# B&R Automation Studio project OpcUaSample410_BrbLibUa103 (part 3)

#### BrbLib.typ - Exported data types
```iecst
(********************************************************************
 * COPYRIGHT -- Bernecker + Rainer
 ********************************************************************
 * Library: BrbLib
 * File: BrbLib.typ
 * Author: niedermeierr
 * Created: June 11, 2013
 ********************************************************************
 * Data types of library BrbLib
 ********************************************************************)
(*Error numbers*)

TYPE
	BrbError_ENUM :
		(
		eBRB_ERR_OK := 0,
		eBRB_ERR_NULL_POINTER := 50000,
		eBRB_ERR_INVALID_PARAMETER := 50001,
		eBRB_ERR_NOT_ENABLED := 50002,
		eBRB_ERR_OVERFLOW := 50003,
		eBRB_ERR_DIVISION_BY_0 := 50004,
		eBRB_ERR_STRING_TOO_SHORT := 50005,
		eBRB_ERR_STRING_TOO_LONG := 50006,
		eBRB_ERR_BUSY := 65535
		);
END_TYPE

(*StepHandling*)

TYPE
	BrbStepHandlingCurrent_TYP : 	STRUCT
		nStepNr : DINT; (*Aktuelle Schrittnummer*)
		sStepText : STRING[nBRB_STEP_TEXT_CHAR_MAX]; (*Aktueller Schritttext*)
		bTimeoutElapsed : BOOL; (*1=Timeout abgelaufen*)
		nTimeoutContinueStep : DINT; (*Schrittnummer nach Timeout*)
	END_STRUCT;
	BrbStepHandlingStep_TYP : 	STRUCT
		nStepNr : DINT; (*Schrittnummer*)
		sStepText : STRING[nBRB_STEP_TEXT_CHAR_MAX]; (*Schritttext*)
		nCycleCount : UDINT; (*Zyklen*)
	END_STRUCT;
	BrbStepHandlingLog_TYP : 	STRUCT
		bClear : BOOL; (*Kommando zum Löschen der Protokollierung*)
		bStop : BOOL; (*Kommando zum Stoppen der Protokollierung*)
		Steps : ARRAY[0..nBRB_STEPLOG_STEPS_MAX]OF BrbStepHandlingStep_TYP; (*Protokollierung*)
	END_STRUCT;
	BrbStepHandlingIntern_TYP : 	STRUCT
		nStepNrOld : DINT; (*Alte Schrittnummer*)
		nCycleCount : UDINT; (*Aktueller Zykluszähler*)
		bLogOnNextCycle : BOOL; (*Flag bei Schrittwechsel*)
		fbTimeout : TON; (*Timeout-Fub*)
	END_STRUCT;
	BrbStepHandling_TYP : 	STRUCT
		Current : BrbStepHandlingCurrent_TYP; (*Daten zum aktuellen Schritt*)
		Log : BrbStepHandlingLog_TYP; (*Protokollierung*)
		Intern : BrbStepHandlingIntern_TYP; (*Interne Daten*)
	END_STRUCT;
	BrbStopWatch_TYP : 	STRUCT
		tStartTime : TIME; (*Start-Zeitstempel*)
		tStopTime : TIME; (*End-Zeitstempel*)
		nTimeDiff : UDINT; (*Berechnete Differenz*)
		sTimeDiff : STRING[24]; (*Differenz als Text*)
	END_STRUCT;
END_TYPE

(*TaskCommunication*)

TYPE
	BrbCallerStates_ENUM :
		(
		eBRB_CALLER_STATE_NOT_READY := -1, (*-1=Nicht bereit*)
		eBRB_CALLER_STATE_OK := 0, (*0=Bereit*)
		eBRB_CALLER_STATE_BUSY := 1 (*1=Besetzt*)
		);
	BrbCaller_TYP : 	STRUCT
		nCallerId : DINT; (*Task-ID*)
		bLock : BOOL; (*Semaphor-Flag*)
	END_STRUCT;
END_TYPE

(*VarHandling*)

TYPE
	BrbLineBreak_ENUM :
		( (*Angabe des Zeilenumbruchs*)
		eBRB_LINE_BREAK_CRLF, (*0=CarriageReturn+LineFeed*)
		eBRB_LINE_BREAK_CR, (*1=CarriageReturn*)
		eBRB_LINE_BREAK_LF (*2=LineFeed*)
		);
	BrbPvInfo_TYP : 	STRUCT
		sName : STRING[nBRB_PVNAME_CHAR_MAX]; (*Variablen-Name*)
		nAdr : UDINT; (*Variablen-Adresse*)
		nDataType : UDINT; (*Variablen-Datentyp*)
		nLen : UDINT; (*Variablen-Größe*)
		nDimension : UINT; (*Max. Array-Index*)
		nItemIndex : UINT; (*Index des Array- oder Struktur-Items*)
	END_STRUCT;
END_TYPE

(*FileHandling*)

TYPE
	BrbUsbDeviceListEntry_TYP : 	STRUCT
		sInterfaceName : STRING[nBRB_DEVICE_NAME_CHAR_MAX]; (*Schnittstellen-Name*)
		sDeviceName : STRING[nBRB_DEVICE_NAME_CHAR_MAX]; (*Schnittstellen-Name*)
		nNode : UDINT; (*Interne Node-Nummer*)
		nHandle : UDINT; (*Internes Handle*)
	END_STRUCT;
	BrbDirInfoFilter_ENUM :
		(
		eBRB_DIR_INFO_ONLY_FILES, (*0=Nur Dateien*)
		eBRB_DIR_INFO_ONLY_DIRS, (*1=Nur Verzeichnisse*)
		eBRB_DIR_INFO_FILES_AND_DIRS (*2=Dateien und Verzeichnisse*)
		);
	BrbFileSorting_ENUM :
		(
		eBRB_FILE_SORTING_NONE, (*0=Keine Sortierung*)
		eBRB_FILE_SORTING_ALPH_UP, (*1=Sortierung nach aufsteigendem Alphabet*)
		eBRB_FILE_SORTING_ALPH_DOWN, (*2=Sortierung nach aufsteigendem Alphabet*)
		eBRB_FILE_SORTING_OLDEST, (*3=Sortierung nach ältesten Dateien*)
		eBRB_FILE_SORTING_YOUNGEST, (*4=Sortierung nach jüngsten Dateien*)
		eBRB_FILE_SORTING_BIGGEST, (*5=Sortierung nach größten Dateien*)
		eBRB_FILE_SORTING_SMALLEST, (*6=Sortierung nach kleinsten Dateien*)
		eBRB_FILE_SORTING_USER (*7=Sortierung mit benutzerdefinierter Vergleichsfunktion*)
		);
	BrbReadDirListEntry_TYP : 	STRUCT
		sName : STRING[nBRB_FILE_NAME_CHAR_MAX]; (*Verzeichnis- oder Datei-Name*)
		dtDate : DATE_AND_TIME; (*Zeitstempel*)
		nSize : UDINT; (*Größe (0=Verzeichnis)*)
	END_STRUCT;
END_TYPE

(*Logger*)

TYPE
	BrbLogHierarchListEntry_TYP : 	STRUCT
		nRecordId : ArEventLogRecordIDType;
		nOriginRecordId : ArEventLogRecordIDType;
		nEventId : DINT;
		nSeverity : USINT;
		sObjectId : STRING[36];
		sDecription : STRING[512];
	END_STRUCT;
	BrbLogHierarchListSevFilter_ENUM :
		(
		eBRB_LOG_SEVERITY_FILTER_ALL := 0, (*Keine Filterung*)
		eBRB_LOG_SEVERITY_FILTER_SUCCESS := 1, (*Nur Erfolgs-Einträge*)
		eBRB_LOG_SEVERITY_FILTER_INFO := 2, (*Nur Info-Einträge*)
		eBRB_LOG_SEVERITY_FILTER_WARNING := 4, (*Nur Warnungs-Einträge*)
		eBRB_LOG_SEVERITY_FILTER_ERROR := 8 (*Nur Fehler-Einträge*)
		);
END_TYPE

(*TimeAndDate*)

TYPE
	BrbWeekdays_ENUM :
		( (*Wochentage*)
		eBRB_WD_SUNDAY, (*0=Sonntag*)
		eBRB_WD_MONDAY, (*1=Montag*)
		eBRB_WD_TUESDAY, (*2=Dienstag*)
		eBRB_WD_WEDNESDAY, (*3=Mittwoch*)
		eBRB_WD_THURSDAY, (*4=Donnerstag*)
		eBRB_WD_FRIDAY, (*5=Freitag*)
		eBRB_WD_SATURDAY (*6=Samstag*)
		);
	BrbTimeAndDateCompare_ENUM :
		(
		eBRB_TAD_COMPARE_YOUNGER,
		eBRB_TAD_COMPARE_YOUNGEREQUAL,
		eBRB_TAD_COMPARE_EQUAL,
		eBRB_TAD_COMPARE_OLDEREQUAL,
		eBRB_TAD_COMPARE_OLDER
		);
	BrbTimerSwitchParTimePoint_TYP : 	STRUCT  (*Schaltpunkt*)
		bActive : BOOL; (*1=Zeitpunkt ist aktiv*)
		dtsTimePoint : DTStructure; (*Zeitpunkt*)
		eSwitchType : BrbTimerSwitchType_ENUM; (*Typ der Schaltung (Aus, An, Umschalten, Puls)*)
	END_STRUCT;
	BrbTimerSwitchPar_TYP : 	STRUCT  (*Parameter der Zeitschaltuhr*)
		eMode : BrbTimerSwitchMode_ENUM; (*Modus der Schaltung (Sekunde, Minute, Stunde...)*)
		TimePoint : ARRAY[0..nBRB_TIMERSWITCH_POINT_INDEX_MAX]OF BrbTimerSwitchParTimePoint_TYP; (*Liste der Schaltpunkte*)
	END_STRUCT;
	BrbTimerSwitchType_ENUM :
		( (*Typ der Schaltung*)
		eBRB_TIMERSWITCH_TYPE_OFF, (*0 = Aus*)
		eBRB_TIMERSWITCH_TYPE_ON, (*1 = An*)
		eBRB_TIMERSWITCH_TYPE_TOGGLE, (*2 = Umschalten*)
		eBRB_TIMERSWITCH_TYPE_IMPULSE (*3 = Puls*)
		);
	BrbTimerSwitchMode_ENUM :
		( (*Modus der Schaltung*)
		eBRB_TIMERSWITCH_MODE_MONTH, (*0=Monat*)
		eBRB_TIMERSWITCH_MODE_WEEK, (*1=Woche*)
		eBRB_TIMERSWITCH_MODE_DAY, (*2=Tag*)
		eBRB_TIMERSWITCH_MODE_HOUR, (*3=Stunde*)
		eBRB_TIMERSWITCH_MODE_MINUTE, (*4=Minute*)
		eBRB_TIMERSWITCH_MODE_SECOND (*5=Sekunde*)
		);
	BrbTimerSwitchWeekdays_ENUM :
		( (*Wochentage*)
		eBRB_TIMERSWITCH_WD_SUNDAY, (*0=Sonntag*)
		eBRB_TIMERSWITCH_WD_MONDAY, (*1=Montag*)
		eBRB_TIMERSWITCH_WD_TUESDAY, (*2=Dienstag*)
		eBRB_TIMERSWITCH_WD_WEDNESDAY, (*3=Mittwoch*)
		eBRB_TIMERSWITCH_WD_THURSDAY, (*4=Donnerstag*)
		eBRB_TIMERSWITCH_WD_FRIDAY, (*5=Freitag*)
		eBRB_TIMERSWITCH_WD_SATURDAY (*6=Samstag*)
		);
END_TYPE

(*BigDataTypes*)

TYPE
	BrbUint64_TYP : 	STRUCT
		nLow : UDINT; (*Niederwertige Bits*)
		nHigh : UDINT; (*Höherwertige Bits*)
	END_STRUCT;
	BrbInt64_TYP : 	STRUCT
		nLow : UDINT; (*Niederwertige Bits*)
		nHigh : UDINT; (*Höherwertige Bits*)
	END_STRUCT;
	BrbDt64Operator_ENUM :
		(
		eBRB_DT64_OPERATOR_ADD,
		eBRB_DT64_OPERATOR_SUBTRACT,
		eBRB_DT64_OPERATOR_MULTIPLY,
		eBRB_DT64_OPERATOR_DIVIDE
		);
END_TYPE

(*Memory*)

TYPE
	BrbMemListManagement_Typ : 	STRUCT
		pList : UDINT; (*Adresse des Array-Anfangs*)
		nEntryLength : UDINT; (*Größe eines Eintrags*)
		nIndexMax : UDINT; (*Maximaler Index des Arrays*)
		nEntryCount : UDINT; (*Momentane Anzahl der gültigen Eintrage*)
	END_STRUCT;
END_TYPE

(*Math*)

TYPE
	BrbRound_ENUM :
		(
		eBRB_ROUND_APPROP, (*Rundung gemäss letzter Stelle(n), Grenze bei 5*)
		eBRB_ROUND_UP, (*Aufrundung*)
		eBRB_ROUND_DOWN (*Abrundung*)
		);
END_TYPE

(*Random*)

TYPE
	BrbRandomString_ENUM :
		(
		eBRB_RANDOM_STRING_NUMBERS := 1, (*Zahler*)
		eBRB_RANDOM_STRING_UPPER_LETTERS := 2, (*Großbuchstaben*)
		eBRB_RANDOM_STRING_LOWER_LETTERS := 4, (*Kleinbuchstaben*)
		eBRB_RANDOM_STRING_SPACE := 8, (*Leerzeichen*)
		eBRB_RANDOM_STRING_PUNCTUATION := 16, (*Satzzeichen*)
		eBRB_RANDOM_STRING_SYMBOLS := 32, (*Symbole*)
		eBRB_RANDOM_STRING_CONTROLCHARS := 64 (*Steuerzeichen*)
		);
END_TYPE

(*IpAndSubnet*)

TYPE
	BrbIpAdrType_ENUM :
		( (*Ip-Adress-Typen*)
		eBRB_IP_ADR_TYPE_UNKNOWN, (*Unbekannte oder ungültige Adresse*)
		eBRB_IP_ADR_TYPE_NETWORK, (*Netzwerk-Adresse*)
		eBRB_IP_ADR_TYPE_HOST, (*Teilnehmer-Adresse*)
		eBRB_IP_ADR_TYPE_BROADCAST (*Broadcast-Adresse*)
		);
END_TYPE

(*Additional*)

TYPE
	BrbCompilerVersion_TYP : 	STRUCT
		bValid : BOOL; (*1=Version konnte ausgelesen werden*)
		nMajor : INT; (*Haupt-Versionsnummer*)
		nMinor : INT; (*Unter-Versionsnummer*)
		nPatch : INT; (*Patch-Versionsnummer*)
		nTotal : DINT; (*Komplette Versionnummer*)
		sText : STRING[10]; (*Versionsnummer als Text*)
	END_STRUCT;
END_TYPE
```

#### BrbLib.var - Exported constants
```iecst
(********************************************************************
 * COPYRIGHT -- Bernecker + Rainer
 ********************************************************************
 * Library: BrbLib
 * File: BrbLib.var
 * Author: niedermeierr
 * Created: June 11, 2013
 ********************************************************************
 * Constants of library BrbLib
 ********************************************************************)
(*General*)
VAR CONSTANT
	nBRB_USINT_MAX : USINT := 255; (*Maximal-Wert eines USINT*)
	nBRB_UINT_MAX : UINT := 65535; (*Maximal-Wert eines UINT*)
	nBRB_UDINT_MAX : UDINT := 4294967295; (*Maximal-Wert eines UDINT*)
	nBRB_SINT_MIN : SINT := -128; (*Minimal-Wert eines SINT*)
	nBRB_SINT_MAX : SINT := 127; (*Maximal-Wert eines SINT*)
	nBRB_INT_MIN : INT := -32768; (*Minimal-Wert eines INT*)
	nBRB_INT_MAX : INT := 32767; (*Maximal-Wert eines INT*)
	nBRB_DINT_MIN : DINT := -2147483648; (*Minimal-Wert eines DINT*)
	nBRB_DINT_MAX : DINT := 2147483647; (*Maximal-Wert eines DINT*)
	nBRB_BITS_PER_BYTE : USINT := 8; (*Anzahl Bits/Byte*)
	sBRB_STX : ARRAY[0..1] OF USINT := [2,0]; (*Start of Text*)
	sBRB_ETX : ARRAY[0..1] OF USINT := [3,0]; (*End of Text*)
	sBRB_TAB : ARRAY[0..1] OF USINT := [9,0]; (*Tabulator*)
	sBRB_LF : ARRAY[0..1] OF USINT := [10,0]; (*LineFeed = Vorschub*)
	sBRB_LFCR : ARRAY[0..2] OF USINT := [10,13,0]; (*LineFeed + CarriageReturn*)
	sBRB_CR : ARRAY[0..1] OF USINT := [13,0]; (*CarriageReturn = Wagenrücklauf*)
	sBRB_CRLF : ARRAY[0..2] OF USINT := [13,10,0]; (*CarriageReturn + LineFeed*)
	sBRB_QM : ARRAY[0..1] OF USINT := [34,0]; (*QuotationMark = Anführungszeichen*)
	sBRB_WC_TAB : ARRAY[0..1] OF UINT := [9,0]; (*Tabulator*)
	sBRB_WC_LF : ARRAY[0..1] OF UINT := [10,0]; (*LineFeed = Vorschub*)
	sBRB_WC_LFCR : ARRAY[0..2] OF UINT := [10,13,0]; (*LineFeed + CarriageReturn*)
	sBRB_WC_CR : ARRAY[0..1] OF UINT := [13,0]; (*CarriageReturn = Wagenrücklauf*)
	sBRB_WC_CRLF : ARRAY[0..2] OF UINT := [13,10,0]; (*CarriageReturn + LineFeed*)
	sBRB_WC_QM : ARRAY[0..1] OF UINT := [34,0]; (*QuotationMark = Anführungszeichen*)
	nBRB_URL_CHAR_MAX : UINT := 300; (*Zeichenanzahl einer URL*)
END_VAR
(*StepHandling*)
VAR CONSTANT
	nBRB_STEP_TEXT_CHAR_MAX : UINT := 50; (*Zeichenanzahl eines Schritt-Textes*)
	nBRB_STEPLOG_STEPS_MAX : UINT := 20; (*Max. Index der Protokollierung*)
END_VAR
(*VarHandling*)
VAR CONSTANT
	nBRB_FILE_LINES_CHAR_MAX : UINT := 50000; (*Zeichenanzahl einer Datei-Zeile*)
	nBRB_PVNAME_CHAR_MAX : UINT := 520; (*Zeichenanzahl eines Prozess-Variablen*)
END_VAR
(*FileHandling*)
VAR CONSTANT
	nBRB_DEVICE_NAME_CHAR_MAX : UDINT := 32; (*Zeichenanzahl eines Laufwerk-Namens*)
	nBRB_FILE_NAME_CHAR_MAX : UDINT := 259; (*Zeichenanzahl eines Datei-Namens*)
	nBRB_USB_DEVICE_LIST_INDEX_MAX : UINT := 5; (*Anzahl der Usb-Devices*)
	nBRB_FILTER_ALL_CHAR_MAX : UDINT := 200; (*Zeichenanzahl einer gesamten Filterangabe*)
	nBRB_FILTER_SINGLE_CHAR_MAX : UDINT := 20; (*Zeichenanzahl einer einzelnen Filterangabe*)
	nBRB_FILTER_SINGLE_INDEX_MAX : UDINT := 10; (*Max. Index der Filterrangaben*)
END_VAR
(*BigDataTypes*)
VAR CONSTANT
	nBRB_UINT64_CHAR_MAX : UINT := 21; (*Zeichenanzahl eines Uint64 (inkl. Null-Terminierung)*)
	nBRB_INT64_CHAR_MAX : UINT := 21; (*Zeichenanzahl eines Int64 (inkl. Null-Terminierung)*)
END_VAR
(*TimeAndDate*)
VAR CONSTANT
	nBRB_HOURS_PER_DAY : UDINT := 24; (*Stunden pro Tag*)
	nBRB_MINUTES_PER_HOUR : UDINT := 60; (*Minuten pro Stunde*)
	nBRB_SECONDS_PER_HOUR : UDINT := 3600; (*Sekunden pro Stunde*)
	nBRB_SECONDS_PER_DAY : UDINT := 86400; (*Sekunden pro Tag*)
	nBRB_SECONDS_PER_MINUTE : UDINT := 60; (*Sekunden pro Minute*)
	nBRB_MILLISECONDS_PER_SECOND : UDINT := 1000; (*Millisekunden pro Sekunde*)
	nBRB_MILLISECONDS_PER_MINUTE : UDINT := 60000; (*Millisekunden pro Minute*)
	nBRB_MILLISECONDS_PER_HOUR : UDINT := 3600000; (*Millisekunden pro Stunde*)
	nBRB_MILLISECONDS_PER_DAY : UDINT := 86400000; (*Millisekunden pro Tag*)
	nBRB_TIME_TEXT_CHAR_MAX : USINT := 24; (*Zeichenanzahl eines Zeitstempels*)
	nBRB_TIMERSWITCH_POINT_INDEX_MAX : UINT := 15; (*Maximaler Index der Zeitpunkt-Liste für die Zeitschaltuhr*)
END_VAR
(*Math*)
VAR CONSTANT
	rBRB_FACTOR_RAD_TO_DEG : REAL := 57.29578; (*Umrechnungsfaktor Bogenmass zu Grad*)
	rBRB_FACTOR_DEG_TO_RAD : REAL := 0.01745329; (*Umrechnungsfaktor Grad zu Bogenmass*)
	rBRB_DEGREE_0 : REAL := 0.0; (*0°*)
	rBRB_DEGREE_90 : REAL := 90.0; (*90°*)
	rBRB_DEGREE_180 : REAL := 180.0; (*180°*)
	rBRB_DEGREE_270 : REAL := 270.0; (*270°*)
	rBRB_DEGREE_360 : REAL := 360.0; (*360°*)
END_VAR
(*IpAndSubnet*)
VAR CONSTANT
	nBRB_IP_ADR_CHAR_MAX : UINT := 16; (*Anzahl der Zeichen einer IP-Adresse*)
END_VAR
```

#### AnsiCFunc.h
```c
/********************************************************************
 * COPYRIGHT -- Bernecker + Rainer
 ********************************************************************
 * Package: Global
 * File: AnsiCFunc.h
 * Author: niedermeierr
 * Created: April 22, 2008
 *******************************************************************/

#include <bur/plctypes.h>

/*
 * stdlib.h
 *
 * Definitions for common types, variables, and functions.
 */

// NOLINTBEGIN(bugprone-reserved-identifier, cert-dcl37-c, cppcoreguidelines-avoid-non-const-global-variables, clang-diagnostic-reserved-identifier)
#ifndef _STDLIB_H_
#define _STDLIB_H_

#include "_ansi.h"

#define __need_size_t
#define __need_wchar_t
#include <stddef.h>

#include <sys/reent.h>
#include <machine/stdlib.h>
#ifndef __STRICT_ANSI__
#include <alloca.h>
#endif

_BEGIN_STD_C

typedef struct
{
  int quot; /* quotient */
  int rem; /* remainder */
} div_t;

typedef struct
{
  long quot; /* quotient */
  long rem; /* remainder */
} ldiv_t;

#ifndef __STRICT_ANSI__
typedef struct
{
  long long int quot; /* quotient */
  long long int rem; /* remainder */
} lldiv_t;
#endif

#ifndef NULL
#define NULL 0
#endif

#define EXIT_FAILURE 1
#define EXIT_SUCCESS 0

#define RAND_MAX __RAND_MAX

extern __IMPORT int __mb_cur_max;

#define MB_CUR_MAX __mb_cur_max

_VOID	_EXFUN(abort,(_VOID) _ATTRIBUTE ((noreturn)));
int	_EXFUN(abs,(int));
int	_EXFUN(atexit,(_VOID (*__func)(_VOID)));
//double	_EXFUN(atof,(const char *__nptr));
#ifndef __STRICT_ANSI__
float	_EXFUN(atoff,(const char *__nptr));
#endif
//int	_EXFUN(atoi,(const char *__nptr));
int	_EXFUN(_atoi_r,(struct _reent *, const char *__nptr));
long	_EXFUN(atol,(const char *__nptr));
long	_EXFUN(_atol_r,(struct _reent *, const char *__nptr));
_PTR	_EXFUN(bsearch,(const _PTR __key,
		       const _PTR __base,
		       size_t __nmemb,
		       size_t __size,
		       int _EXPARM(_compar,(const _PTR, const _PTR))));
_PTR	_EXFUN(calloc,(size_t __nmemb, size_t __size));
div_t	_EXFUN(div,(int __numer, int __denom));
_VOID	_EXFUN(exit,(int __status) _ATTRIBUTE ((noreturn)));
_VOID	_EXFUN(free,(_PTR));
char *  _EXFUN(getenv,(const char *__string));
char *	_EXFUN(_getenv_r,(struct _reent *, const char *__string));
#ifdef __CYGWIN__
const char *_EXFUN(getprogname,(void));
#endif
char *	_EXFUN(_findenv,(_CONST char *, int *));
char *	_EXFUN(_findenv_r,(struct _reent *, _CONST char *, int *));
long	_EXFUN(labs,(long));
ldiv_t	_EXFUN(ldiv,(long __numer, long __denom));
_PTR	_EXFUN(malloc,(size_t __size));
int	_EXFUN(mblen,(const char *, size_t));
int	_EXFUN(_mblen_r,(struct _reent *, const char *, size_t, _mbstate_t *));
int	_EXFUN(mbtowc,(wchar_t *, const char *, size_t));
int	_EXFUN(_mbtowc_r,(struct _reent *, wchar_t *, const char *, size_t, _mbstate_t *));
int	_EXFUN(wctomb,(char *, wchar_t));
int	_EXFUN(_wctomb_r,(struct _reent *, char *, wchar_t, _mbstate_t *));
size_t	_EXFUN(mbstowcs,(wchar_t *, const char *, size_t));
size_t	_EXFUN(_mbstowcs_r,(struct _reent *, wchar_t *, const char *, size_t, _mbstate_t *));
size_t	_EXFUN(wcstombs,(char *, const wchar_t *, size_t));
size_t	_EXFUN(_wcstombs_r,(struct _reent *, char *, const wchar_t *, size_t, _mbstate_t *));
#ifndef __STRICT_ANSI__
#ifndef _REENT_ONLY
int     _EXFUN(mkstemp,(char *));
char *  _EXFUN(mktemp,(char *));
#endif
#endif
_VOID	_EXFUN(qsort,(_PTR __base, size_t __nmemb, size_t __size, int(*_compar)(const _PTR, const _PTR)));
int	_EXFUN(rand,(_VOID));
_PTR	_EXFUN(realloc,(_PTR __r, size_t __size));
#ifdef __CYGWIN__
void	_EXFUN(setprogname,(const char *));
#endif
_VOID	_EXFUN(srand,(unsigned __seed));
double	_EXFUN(strtod,(const char *__n, char **__end_PTR));
double	_EXFUN(_strtod_r,(struct _reent *,const char *__n, char **__end_PTR));
float	_EXFUN(strtof,(const char *__n, char **__end_PTR));
#ifndef __STRICT_ANSI__
/* the following strtodf interface is deprecated...use strtof instead */
# ifndef strtodf
#  define strtodf strtof
# endif
#endif
long	_EXFUN(strtol,(const char *__n, char **__end_PTR, int __base));
long	_EXFUN(_strtol_r,(struct _reent *,const char *__n, char **__end_PTR, int __base));
unsigned long _EXFUN(strtoul,(const char *__n, char **__end_PTR, int __base));
unsigned long _EXFUN(_strtoul_r,(struct _reent *,const char *__n, char **__end_PTR, int __base));

int	_EXFUN(system,(const char *__string));

#ifndef __STRICT_ANSI__
long    _EXFUN(a64l,(const char *__input));
char *  _EXFUN(l64a,(long __input));
char *  _EXFUN(_l64a_r,(struct _reent *,long __input));
int	_EXFUN(on_exit,(_VOID (*__func)(int, _PTR),_PTR __arg));
_VOID	_EXFUN(_Exit,(int __status) _ATTRIBUTE ((noreturn)));
int	_EXFUN(putenv,(const char *__string));
int	_EXFUN(_putenv_r,(struct _reent *, const char *__string));
int	_EXFUN(setenv,(const char *__string, const char *__value, int __overwrite));
int	_EXFUN(_setenv_r,(struct _reent *, const char *__string, const char *__value, int __overwrite));

char *	_EXFUN(gcvt,(double,int,char *));
char *	_EXFUN(gcvtf,(float,int,char *));
char *	_EXFUN(fcvt,(double,int,int *,int *));
char *	_EXFUN(fcvtf,(float,int,int *,int *));
char *	_EXFUN(ecvt,(double,int,int *,int *));
char *	_EXFUN(ecvtbuf,(double, int, int*, int*, char *));
char *	_EXFUN(fcvtbuf,(double, int, int*, int*, char *));
char *	_EXFUN(ecvtf,(float,int,int *,int *));
char *	_EXFUN(dtoa,(double, int, int, int *, int*, char**));
int	_EXFUN(rand_r,(unsigned *__seed));

double _EXFUN(drand48,(_VOID));
double _EXFUN(_drand48_r,(struct _reent *));
double _EXFUN(erand48,(unsigned short [3]));
double _EXFUN(_erand48_r,(struct _reent *, unsigned short [3]));
long   _EXFUN(jrand48,(unsigned short [3]));
long   _EXFUN(_jrand48_r,(struct _reent *, unsigned short [3]));
_VOID  _EXFUN(lcong48,(unsigned short [7]));
_VOID  _EXFUN(_lcong48_r,(struct _reent *, unsigned short [7]));
long   _EXFUN(lrand48,(_VOID));
long   _EXFUN(_lrand48_r,(struct _reent *));
long   _EXFUN(mrand48,(_VOID));
long   _EXFUN(_mrand48_r,(struct _reent *));
long   _EXFUN(nrand48,(unsigned short [3]));
long   _EXFUN(_nrand48_r,(struct _reent *, unsigned short [3]));
unsigned short *
       _EXFUN(seed48,(unsigned short [3]));
unsigned short *
       _EXFUN(_seed48_r,(struct _reent *, unsigned short [3]));
_VOID  _EXFUN(srand48,(long));
_VOID  _EXFUN(_srand48_r,(struct _reent *, long));
long long _EXFUN(atoll,(const char *__nptr));
long long _EXFUN(_atoll_r,(struct _reent *, const char *__nptr));
long long _EXFUN(llabs,(long long));
lldiv_t	_EXFUN(lldiv,(long long __numer, long long __denom));
long long _EXFUN(strtoll,(const char *__n, char **__end_PTR, int __base));
long long _EXFUN(_strtoll_r,(struct _reent *, const char *__n, char **__end_PTR, int __base));
unsigned long long _EXFUN(strtoull,(const char *__n, char **__end_PTR, int __base));
unsigned long long _EXFUN(_strtoull_r,(struct _reent *, const char *__n, char **__end_PTR, int __base));

#ifndef __CYGWIN__
_VOID	_EXFUN(cfree,(_PTR));
#else
char *	_EXFUN(realpath,(const char *, char *));
void	_EXFUN(unsetenv,(const char *__string));
void	_EXFUN(_unsetenv_r,(struct _reent *, const char *__string));
int	_EXFUN(random,(_VOID));
long	_EXFUN(srandom,(unsigned __seed));
char *  _EXFUN(ptsname, (int));
int     _EXFUN(grantpt, (int));
int     _EXFUN(unlockpt,(int));
#endif

#endif /* ! __STRICT_ANSI__ */

char *	_EXFUN(_dtoa_r,(struct _reent *, double, int, int, int *, int*, char**));
#ifndef __CYGWIN__
_PTR	_EXFUN(_malloc_r,(struct _reent *, size_t));
_PTR	_EXFUN(_calloc_r,(struct _reent *, size_t, size_t));
_VOID	_EXFUN(_free_r,(struct _reent *, _PTR));
_PTR	_EXFUN(_realloc_r,(struct _reent *, _PTR, size_t));
_VOID	_EXFUN(_mstats_r,(struct _reent *, char *));
#endif
int	_EXFUN(_system_r,(struct _reent *, const char *));

_VOID	_EXFUN(__eprintf,(const char *, const char *, unsigned int, const char *));

#ifdef __CYGWIN__
#undef _malloc_r
#define _malloc_r(r, s) malloc (s)
#undef _free_r
#define _free_r(r, p) free (p)
#undef _realloc_r
#define _realloc_r(r, p, s) realloc (p, s)
#undef _calloc_r
#define _calloc_r(r, s1, s2) calloc (s1, s2);
#undef _memalign_r
#define _memalign_r(r, s1, s2) memalign (s1, s2);
#undef _mallinfo_r
#define _mallinfo_r(r) mallinfo ()
#undef _malloc_stats_r
#define _malloc_stats_r(r) malloc_stats ()
#undef _mallopt_r
#define _mallopt_r(i1, i2) mallopt (i1, i2)
#undef _malloc_usable_size_r
#define _malloc_usable_size_r(r, p) malloc_usable_size (p)
#undef _valloc_r
#define _valloc_r(r, s) valloc (s)
#undef _pvalloc_r
#define _pvalloc_r(r, s) pvalloc (s)
#undef _malloc_trim_r
#define _malloc_trim_r(r, s) malloc_trim (s)
#undef _mstats_r
#define _mstats_r(r, p) mstats (p)
#endif

_END_STD_C

#endif /* _STDLIB_H_ */
// NOLINTEND(bugprone-reserved-identifier, cert-dcl37-c, cppcoreguidelines-avoid-non-const-global-variables, clang-diagnostic-reserved-identifier)
```

#### Package Logical/Libraries/BrbLib/StepHandling - Schrittketten-Behandlung

#### BrbStartStepTimeout.c
```c
/********************************************************************
 * COPYRIGHT -- Bernecker + Rainer
 ********************************************************************
 * Library: BrbLib
 * File: BrbStartStepTimeout.c
 * Author: niedermeierr
 * Created: June 11, 2013
 ********************************************************************
 * Implementation of library BrbLib
 ********************************************************************/

#include <bur/plctypes.h>
#ifdef __cplusplus
	extern "C"
	{
#endif

#include "BrbLib.h"

#ifdef __cplusplus
	};
#endif

 // NOLINTBEGIN(readability-*, bugprone-easily-swappable-parameters, clang-diagnostic-invalid-utf8, clang-diagnostic-invalid-source-encoding, clang-diagnostic-pointer-arith, clang-diagnostic-strict-prototypes, hicpp-uppercase-literal-suffix, cppcoreguidelines-*, performance-*)

/* Startet den Timeout-Zähler für eine Schrittkette */
unsigned short BrbStartStepTimeout(struct BrbStepHandling_TYP* pStepHandling, unsigned long nTimeout, signed long nContinueStep)
{
	// Prüfen, ob Timer schon abgelaufen ist
	if(pStepHandling->Intern.fbTimeout.Q == 0)
	{
		// Timer setzen und starten
		pStepHandling->Intern.fbTimeout.PT = (TIME)nTimeout;
		pStepHandling->Current.nTimeoutContinueStep = nContinueStep;
		pStepHandling->Intern.fbTimeout.IN = 1;
	}
	return 0;
}

// NOLINTEND(readability-*, bugprone-easily-swappable-parameters, clang-diagnostic-invalid-utf8, clang-diagnostic-invalid-source-encoding, clang-diagnostic-pointer-arith, clang-diagnostic-strict-prototypes, hicpp-uppercase-literal-suffix, cppcoreguidelines-*, performance-*)
```

#### BrbStartStopWatch.c
```c
/********************************************************************
 * COPYRIGHT -- Bernecker + Rainer
 ********************************************************************
 * Library: BrbLib
 * File: BrbStartStopWatch.c
 * Author: niedermeierr
 * Created: June 11, 2013
 ********************************************************************
 * Implementation of library BrbLib
 ********************************************************************/

#include <bur/plctypes.h>
#ifdef __cplusplus
	extern "C"
	{
#endif

#include "BrbLib.h"
#include <string.h>

#ifdef __cplusplus
	};
#endif

// NOLINTBEGIN(readability-*, bugprone-easily-swappable-parameters, clang-diagnostic-invalid-utf8, clang-diagnostic-invalid-source-encoding, clang-diagnostic-pointer-arith, clang-diagnostic-strict-prototypes, hicpp-uppercase-literal-suffix, cppcoreguidelines-*, performance-*)

/* Startet eine Stoppuhr */
plcbit BrbStartStopWatch(struct BrbStopWatch_TYP* pStopWatch)
{
	// Stoppuhr starten
	pStopWatch->tStartTime = clock_ms();
	pStopWatch->nTimeDiff = 0;
	memset(pStopWatch->sTimeDiff, 0, sizeof(pStopWatch->sTimeDiff));
	return 0;
}

// NOLINTEND(readability-*, bugprone-easily-swappable-parameters, clang-diagnostic-invalid-utf8, clang-diagnostic-invalid-source-encoding, clang-diagnostic-pointer-arith, clang-diagnostic-strict-prototypes, hicpp-uppercase-literal-suffix, cppcoreguidelines-*, performance-*)
```

#### BrbStepHandler.c
```c
/********************************************************************
 * COPYRIGHT -- Bernecker + Rainer
 ********************************************************************
 * Library: BrbLib
 * File: BrbStepHandler.c
 * Author: niedermeierr
 * Created: June 11, 2013
 ********************************************************************
 * Implementation of library BrbLib
 ********************************************************************/

#include <bur/plctypes.h>
#ifdef __cplusplus
	extern "C"
	{
#endif

#include "BrbLib.h"
#include <string.h>

#ifdef __cplusplus
	};
#endif

 // NOLINTBEGIN(readability-*, bugprone-easily-swappable-parameters, clang-diagnostic-invalid-utf8, clang-diagnostic-invalid-source-encoding, clang-diagnostic-pointer-arith, clang-diagnostic-strict-prototypes, hicpp-uppercase-literal-suffix, cppcoreguidelines-*, performance-*)

/* Behandelt Schrittketten (Protokollierung, Timeout usw.) */
signed long BrbStepHandler(struct BrbStepHandling_TYP* pStepHandling)
{
	// Muss der Schritt protokolliert werden?
	if(pStepHandling->Intern.bLogOnNextCycle == 1)
	{
		pStepHandling->Intern.bLogOnNextCycle = 0;
		// Ist Protokollierung gestoppt?
		if(pStepHandling->Log.bStop == 0)
		{
			// Zykluszähler merken
			pStepHandling->Log.Steps[0].nCycleCount = pStepHandling->Intern.nCycleCount;
			// Einträge um eins nach unten schieben
			memmove(&pStepHandling->Log.Steps[1], &pStepHandling->Log.Steps[0], sizeof(BrbStepHandlingStep_TYP)*(nBRB_STEPLOG_STEPS_MAX));
			// Aktuellen Eintrag reinkopieren
			pStepHandling->Log.Steps[0].nStepNr = pStepHandling->Intern.nStepNrOld;
			BrbStringCopy(pStepHandling->Log.Steps[0].sStepText, pStepHandling->Current.sStepText, sizeof(pStepHandling->Log.Steps[0].sStepText));
		}
		// Zykluszähler wieder auf 0 setzen
		pStepHandling->Intern.nCycleCount = 0;
	}
	// Hat sich der Schritt geändert?
	if(pStepHandling->Current.nStepNr != pStepHandling->Intern.nStepNrOld)
	{
		// Schritt beim nächsten Durchlauf protokollieren, weil dann erst der richtige Schritttext gesetzt ist
		pStepHandling->Intern.bLogOnNextCycle = 1;
	}
	// Zykluszähler erhöhen
	pStepHandling->Intern.nCycleCount++;
	// Aktuellen Schritt übernehmen
	pStepHandling->Intern.nStepNrOld = pStepHandling->Current.nStepNr;
	// Kommando zum Löschen der Protokollierung
	if(pStepHandling->Log.bClear == 1)
	{
		pStepHandling->Log.bClear = 0;
		// Den gesamten Aufzeichnungspuffer löschen
		memset(&pStepHandling->Log.Steps[0], 0, sizeof(pStepHandling->Log.Steps));
		pStepHandling->Intern.bLogOnNextCycle = 1;
	}
	// StepTimeout
	TON(&pStepHandling->Intern.fbTimeout);
	if(pStepHandling->Intern.fbTimeout.Q == 1)
	{
		// Timeout abgelaufen
		pStepHandling->Intern.fbTimeout.IN = 0;
		pStepHandling->Current.bTimeoutElapsed = 1;
	}
	return eBRB_ERR_OK;
}

 // NOLINTEND(readability-*, bugprone-easily-swappable-parameters, clang-diagnostic-invalid-utf8, clang-diagnostic-invalid-source-encoding, clang-diagnostic-pointer-arith, clang-diagnostic-strict-prototypes, hicpp-uppercase-literal-suffix, cppcoreguidelines-*, performance-*)
```

#### BrbStopStepTimeout.c
```c
/********************************************************************
 * COPYRIGHT -- Bernecker + Rainer
 ********************************************************************
 * Library: BrbLib
 * File: BrbStopStepTimeout.c
 * Author: niedermeierr
 * Created: June 11, 2013
 ********************************************************************
 * Implementation of library BrbLib
 ********************************************************************/

#include <bur/plctypes.h>
#ifdef __cplusplus
	extern "C"
	{
#endif

#include "BrbLib.h"

#ifdef __cplusplus
	};
#endif

// NOLINTBEGIN(readability-*, bugprone-easily-swappable-parameters, clang-diagnostic-invalid-utf8, clang-diagnostic-invalid-source-encoding, clang-diagnostic-pointer-arith, clang-diagnostic-strict-prototypes, hicpp-uppercase-literal-suffix, cppcoreguidelines-*, performance-*)

/* Stoppt den Timeout-Zähler für eine Schrittkette */
unsigned short BrbStopStepTimeout(struct BrbStepHandling_TYP* pStepHandling)
{
	// Timer stoppen
	pStepHandling->Intern.fbTimeout.IN = 0;
	return 0;
}

// NOLINTEND(readability-*, bugprone-easily-swappable-parameters, clang-diagnostic-invalid-utf8, clang-diagnostic-invalid-source-encoding, clang-diagnostic-pointer-arith, clang-diagnostic-strict-prototypes, hicpp-uppercase-literal-suffix, cppcoreguidelines-*, performance-*)
```

#### BrbStopStopWatch.c
```c
/********************************************************************
 * COPYRIGHT -- Bernecker + Rainer
 ********************************************************************
 * Library: BrbLib
 * File: BrbStopStopWatch.c
 * Author: niedermeierr
 * Created: June 11, 2013
 ********************************************************************
 * Implementation of library BrbLib
 ********************************************************************/

#include <bur/plctypes.h>
#ifdef __cplusplus
	extern "C"
	{
#endif

#include "BrbLib.h"
#include <string.h>

#ifdef __cplusplus
	};
#endif

// NOLINTBEGIN(readability-*, bugprone-easily-swappable-parameters, clang-diagnostic-invalid-utf8, clang-diagnostic-invalid-source-encoding, clang-diagnostic-pointer-arith, clang-diagnostic-strict-prototypes, hicpp-uppercase-literal-suffix, cppcoreguidelines-*, performance-*)

/* Stoppt eine Stoppuhr */
unsigned long BrbStopStopWatch(struct BrbStopWatch_TYP* pStopWatch)
{
	// Stoppuhr stoppen
	pStopWatch->tStopTime = clock_ms();
	pStopWatch->nTimeDiff = DiffT(pStopWatch->tStopTime, pStopWatch->tStartTime);
	memset(pStopWatch->sTimeDiff, 0, sizeof(pStopWatch->sTimeDiff));
	TIMEStructure TimeDiff;
	TIME_TO_TIMEStructure((TIME)pStopWatch->nTimeDiff, (UDINT)&TimeDiff);
	STRING sItoA[20];
	memset(sItoA, 0, sizeof(sItoA));
	if(TimeDiff.day < 10)
	{
		BrbStringCat((STRING*)pStopWatch->sTimeDiff, "0", sizeof(pStopWatch->sTimeDiff));
	}
	brsitoa((DINT)TimeDiff.day, (UDINT)&sItoA);
	BrbStringCat((STRING*)pStopWatch->sTimeDiff, sItoA, sizeof(pStopWatch->sTimeDiff));
	BrbStringCat((STRING*)pStopWatch->sTimeDiff, "d_", sizeof(pStopWatch->sTimeDiff));
	if(TimeDiff.hour < 10)
	{
		BrbStringCat((STRING*)pStopWatch->sTimeDiff, "0", sizeof(pStopWatch->sTimeDiff));
	}
	brsitoa((DINT)TimeDiff.hour, (UDINT)&sItoA);
	BrbStringCat((STRING*)pStopWatch->sTimeDiff, sItoA, sizeof(pStopWatch->sTimeDiff));
	BrbStringCat((STRING*)pStopWatch->sTimeDiff, "h_", sizeof(pStopWatch->sTimeDiff));
	if(TimeDiff.minute < 10)
	{
		BrbStringCat((STRING*)pStopWatch->sTimeDiff, "0", sizeof(pStopWatch->sTimeDiff));
	}
	brsitoa((DINT)TimeDiff.minute, (UDINT)&sItoA);
	BrbStringCat((STRING*)pStopWatch->sTimeDiff, sItoA, sizeof(pStopWatch->sTimeDiff));
	BrbStringCat((STRING*)pStopWatch->sTimeDiff, "m_", sizeof(pStopWatch->sTimeDiff));
	if(TimeDiff.second < 10)
	{
		BrbStringCat((STRING*)pStopWatch->sTimeDiff, "0", sizeof(pStopWatch->sTimeDiff));
	}
	brsitoa((DINT)TimeDiff.second, (UDINT)&sItoA);
	BrbStringCat((STRING*)pStopWatch->sTimeDiff, sItoA, sizeof(pStopWatch->sTimeDiff));
	BrbStringCat((STRING*)pStopWatch->sTimeDiff, "s_", sizeof(pStopWatch->sTimeDiff));
	if(TimeDiff.millisec < 10)
	{
		BrbStringCat((STRING*)pStopWatch->sTimeDiff, "00", sizeof(pStopWatch->sTimeDiff));
	}
	else if(TimeDiff.millisec < 100)
	{
		BrbStringCat((STRING*)pStopWatch->sTimeDiff, "0", sizeof(pStopWatch->sTimeDiff));
	}
	brsitoa((DINT)TimeDiff.millisec, (UDINT)&sItoA);
	BrbStringCat((STRING*)pStopWatch->sTimeDiff, sItoA, sizeof(pStopWatch->sTimeDiff));
	BrbStringCat((STRING*)pStopWatch->sTimeDiff, "ms", sizeof(pStopWatch->sTimeDiff));
	return pStopWatch->nTimeDiff;
}

// NOLINTEND(readability-*, bugprone-easily-swappable-parameters, clang-diagnostic-invalid-utf8, clang-diagnostic-invalid-source-encoding, clang-diagnostic-pointer-arith, clang-diagnostic-strict-prototypes, hicpp-uppercase-literal-suffix, cppcoreguidelines-*, performance-*)
```

#### Package Logical/Libraries/BrbLib/TaskCommunication - Task-Kommunikation

#### BrbClearCallerBox.c
```c
/********************************************************************
 * COPYRIGHT -- Bernecker + Rainer
 ********************************************************************
 * Library: BrbLib
 * File: BrbClearCallerBox.c
 * Author: niedermeierr
 * Created: June 11, 2013
 ********************************************************************
 * Implementation of library BrbLib
 ********************************************************************/

#include <bur/plctypes.h>
#ifdef __cplusplus
	extern "C"
	{
#endif

#include "BrbLib.h"
#include <string.h>

#ifdef __cplusplus
	};
#endif

// NOLINTBEGIN(readability-*, bugprone-easily-swappable-parameters, clang-diagnostic-invalid-utf8, clang-diagnostic-invalid-source-encoding, clang-diagnostic-pointer-arith, clang-diagnostic-strict-prototypes, hicpp-uppercase-literal-suffix, cppcoreguidelines-*, performance-*)

/* Setzt eine CallerBox komplett auf 0 */
unsigned short BrbClearCallerBox(unsigned long pCallerBox, unsigned long nSize)
{
	memset((USINT*)pCallerBox, 0, nSize);
	return eBRB_ERR_OK;
}

// NOLINTEND(readability-*, bugprone-easily-swappable-parameters, clang-diagnostic-invalid-utf8, clang-diagnostic-invalid-source-encoding, clang-diagnostic-pointer-arith, clang-diagnostic-strict-prototypes, hicpp-uppercase-literal-suffix, cppcoreguidelines-*, performance-*)
```

#### BrbClearDirectBox.c
```c
/********************************************************************
 * COPYRIGHT -- Bernecker + Rainer
 ********************************************************************
 * Library: BrbLib
 * File: BrbClearDirectBox.c
 * Author: niedermeierr
 * Created: June 11, 2013
 ********************************************************************
 * Implementation of library BrbLib
 ********************************************************************/

#include <bur/plctypes.h>
#ifdef __cplusplus
	extern "C"
	{
#endif

#include "BrbLib.h"
#include <string.h>

#ifdef __cplusplus
	};
#endif

// NOLINTBEGIN(readability-*, bugprone-easily-swappable-parameters, clang-diagnostic-invalid-utf8, clang-diagnostic-invalid-source-encoding, clang-diagnostic-pointer-arith, clang-diagnostic-strict-prototypes, hicpp-uppercase-literal-suffix, cppcoreguidelines-*, performance-*)

/* Setzt eine DirectBox komplett auf 0 */
unsigned short BrbClearDirectBox(unsigned long pDirectBox, unsigned long nSize)
{
	memset((USINT*)pDirectBox, 0, nSize);
	return eBRB_ERR_OK;
}

// NOLINTEND(readability-*, bugprone-easily-swappable-parameters, clang-diagnostic-invalid-utf8, clang-diagnostic-invalid-source-encoding, clang-diagnostic-pointer-arith, clang-diagnostic-strict-prototypes, hicpp-uppercase-literal-suffix, cppcoreguidelines-*, performance-*)
```

#### BrbSetCaller.c
```c
/********************************************************************
 * COPYRIGHT -- Bernecker + Rainer
 ********************************************************************
 * Library: BrbLib
 * File: BrbSetCaller.c
 * Author: niedermeierr
 * Created: June 11, 2013
 ********************************************************************
 * Implementation of library BrbLib
 ********************************************************************/

#include <bur/plctypes.h>
#ifdef __cplusplus
	extern "C"
	{
#endif

#include "BrbLib.h"

#ifdef __cplusplus
	};
#endif

// NOLINTBEGIN(readability-*, bugprone-easily-swappable-parameters, clang-diagnostic-invalid-utf8, clang-diagnostic-invalid-source-encoding, clang-diagnostic-pointer-arith, clang-diagnostic-strict-prototypes, hicpp-uppercase-literal-suffix, cppcoreguidelines-*, performance-*)

/* Versucht, die Reservierung für ein Task-Kommando zu erhalten */
BrbCallerStates_ENUM BrbSetCaller(struct BrbCaller_TYP* pCaller, signed long nCallerId)
{
	// Prüfung der Parameter
	if(pCaller == 0)
	{
		return eBRB_CALLER_STATE_NOT_READY;
	}
	// Prüfen, ob die CallerId gesetzt werden kann
	if((pCaller->nCallerId == 0) && (pCaller->bLock == 0))
	{
		// CallerId setzen
		pCaller->nCallerId = nCallerId;
		// Prüfen, ob der Aufruf von einer schnelleren Taskklasse unterbrochen wurde
		if((pCaller->nCallerId == nCallerId) && (pCaller->bLock == 0))
		{
			// CallerId konnte gesetzt werden
			pCaller->bLock = 1;
			return eBRB_CALLER_STATE_OK;
		}
		else
		{
			// Das Setzen wurde von einer schnelleren Taskklasse unterbrochen
			return eBRB_CALLER_STATE_BUSY;
		}
	}
	else if(pCaller->nCallerId == -1)
	{
		// Der Task ist noch nicht bereit
		return eBRB_CALLER_STATE_NOT_READY;
	}
	else
	{
		// Der Task ist schon reserviert
		return eBRB_CALLER_STATE_BUSY;
	}
}

// NOLINTEND(readability-*, bugprone-easily-swappable-parameters, clang-diagnostic-invalid-utf8, clang-diagnostic-invalid-source-encoding, clang-diagnostic-pointer-arith, clang-diagnostic-strict-prototypes, hicpp-uppercase-literal-suffix, cppcoreguidelines-*, performance-*)
```

#### Package Logical/Libraries/BrbLib/VarHandling - Variablen-Funktionen

#### BrbLoadVarAscii.c
```c
/********************************************************************
 * COPYRIGHT -- Bernecker + Rainer
 ********************************************************************
 * Library: BrbLib
 * File: BrbLoadVarAscii.c
 * Author: niedermeierr
 * Created: June 11, 2013
 ********************************************************************
 * Implementation of library BrbLib
 ********************************************************************/

#include <bur/plctypes.h>
#ifdef __cplusplus
	extern "C"
	{
#endif

#include "BrbLib.h"
#include <string.h>

#ifdef __cplusplus
	};
#endif

// NOLINTBEGIN(readability-*, bugprone-easily-swappable-parameters, clang-diagnostic-invalid-utf8, clang-diagnostic-invalid-source-encoding, clang-diagnostic-pointer-arith, clang-diagnostic-strict-prototypes, hicpp-uppercase-literal-suffix, cppcoreguidelines-*, performance-*)

// Eigene Enums und Typen
enum Steps_ENUM
{
	eSTEP_INIT,
	eSTEP_GET_DATAOBJ_INFO,
	eSTEP_DELETE_DATAOBJ_START,
	eSTEP_OPEN_FILE,
	eSTEP_CREATE_DATAOBJ,
	eSTEP_READ_FILE,
	eSTEP_CLOSE_FILE,
	eSTEP_READ_LINES,
	eSTEP_DELETE_DATAOBJ_END,
};

enum Datatypes_ENUM
{
	eDATATYPE_STRUCT,
	eDATATYPE_BOOL,
	eDATATYPE_SINT,
	eDATATYPE_INT,
	eDATATYPE_DINT,
	eDATATYPE_USINT,
	eDATATYPE_UINT,
	eDATATYPE_UDINT,
	eDATATYPE_REAL,
	eDATATYPE_STRING,
	eDATATYPE_DATE_AND_TIME = 11,
	eDATATYPE_TIME,
	eDATATYPE_STRUCT_ARRAY = 15
};

// Prototypen
STRING* SetToNextLine(STRING* pText, STRING* pTextEnd, STRING* pLineBreak);
STRING* ReadPvName(STRING* pText, STRING* pPvName, STRING* pTextEnd);
STRING* ReadPvValue(STRING* pText, STRING* pPvValue, STRING* pTextEnd);
void SetValue(BrbPvInfo_TYP* pPvInfo, STRING* pValue);

/* Lädt eine Ascii-Datei mit Variablen-Werten */
void BrbLoadVarAscii(struct BrbLoadVarAscii* inst) // NOLINT(readability-function-cognitive-complexity)
{
	// Prüfung der Parameter
	if(inst->pDevice == 0)
	{
		inst->nStatus = eBRB_ERR_NULL_POINTER;
		return;
	}
	if(inst->pFile == 0)
	{
		inst->nStatus = eBRB_ERR_NULL_POINTER;
		return;
	}

	switch(inst->eStep)
	{
		case eSTEP_INIT:
			// Fub initialisieren
			inst->nStatus = eBRB_ERR_BUSY;
			inst->nStatusIntern = 0;
			memset(&inst->fbDatObjInfo, 0, sizeof(inst->fbDatObjInfo));
			memset(&inst->fbDatObjDelete, 0, sizeof(inst->fbDatObjDelete));
			memset(&inst->fbFileOpen, 0, sizeof(inst->fbFileOpen));
			memset(&inst->fbDatObjCreate, 0, sizeof(inst->fbDatObjCreate));
			switch(inst->eLineBeak) // NOLINT(clang-diagnostic-switch-enum)
			{
				case eBRB_LINE_BREAK_CR:
					strcpy(inst->sLineBreak, "\r");
					break;
				case eBRB_LINE_BREAK_LF:
					strcpy(inst->sLineBreak, "\n");
					break;
				default:
					strcpy(inst->sLineBreak, "\r\n");
					break;
			}
			if(inst->nLinesToReadAtOneStep == 0)
			{
				// Wenn keine Anzahl angegeben ist, einen Defaultwert verwenden
				inst->nLinesToReadAtOneStep = 10;
			}
			inst->pTextStart = 0;
			inst->pTextEnd = 0;
			inst->pText = 0;
			inst->nLineCountRead = 0;
			memset(&inst->fbFileRead, 0, sizeof(inst->fbFileRead));
			memset(&inst->fbFileClose, 0, sizeof(inst->fbFileClose));
			inst->eStep = eSTEP_GET_DATAOBJ_INFO;
			break;

		case eSTEP_GET_DATAOBJ_INFO:
			// Prüfen, ob noch ein altes Datenobjekt vorhanden ist
			inst->nStatus = eBRB_ERR_BUSY;
			inst->fbDatObjInfo.enable = 1;
			inst->fbDatObjInfo.pName = (UDINT)&"LdPv123";
			DatObjInfo(&inst->fbDatObjInfo);
			if(inst->fbDatObjInfo.status == 0)
			{
				// Vorhanden -> löschen
				inst->eStep = eSTEP_DELETE_DATAOBJ_START;
			}
			else if(inst->fbDatObjInfo.status != eBRB_ERR_BUSY)
			{
				// Nicht vorhanden -> Datei öffnen
				inst->eStep = eSTEP_OPEN_FILE;
			}
			break;

		case eSTEP_DELETE_DATAOBJ_START:
			// Evtl. noch vorhandenes Datenobjekt löschen
			inst->nStatus = eBRB_ERR_BUSY;
			inst->fbDatObjDelete.enable = 1;
			inst->fbDatObjDelete.ident = inst->fbDatObjCreate.ident;
			DatObjDelete(&inst->fbDatObjDelete);
			if(inst->fbDatObjDelete.status == 0)
			{
				inst->eStep = eSTEP_OPEN_FILE;
			}
			else if(inst->fbDatObjDelete.status != eBRB_ERR_BUSY)
			{
				inst->nStatus = inst->fbFileOpen.status;
				inst->eStep = eSTEP_INIT;
			}
			break;

		case eSTEP_OPEN_FILE:
			// Datei öffnen
			inst->nStatus = eBRB_ERR_BUSY;
			inst->fbFileOpen.enable = 1;
			inst->fbFileOpen.pDevice = (UDINT)inst->pDevice;
			inst->fbFileOpen.pFile = (UDINT)inst->pFile;
			FileOpen(&inst->fbFileOpen);
			if(inst->fbFileOpen.status == 0)
			{
				inst->eStep = eSTEP_CREATE_DATAOBJ;
			}
			else if(inst->fbFileOpen.status != eBRB_ERR_BUSY)
			{
				inst->nStatus = inst->fbFileOpen.status;
				inst->eStep = eSTEP_INIT;
			}
			break;

		case eSTEP_CREATE_DATAOBJ:
			// Datenobjekt mit der Größe der Datei erzeugen
			inst->nStatus = eBRB_ERR_BUSY;
			inst->fbDatObjCreate.enable = 1;
			inst->fbDatObjCreate.grp = 0;
			inst->fbDatObjCreate.pName = (UDINT)&"LdPv123";
			inst->fbDatObjCreate.len = inst->fbFileOpen.filelen;
			inst->fbDatObjCreate.MemType = doTEMP;
			inst->fbDatObjCreate.Option = doNO_CS;
			inst->fbDatObjCreate.pCpyData = 0;
			DatObjCreate(&inst->fbDatObjCreate);
			if(inst->fbDatObjCreate.status == 0)
			{
				inst->pTextStart = (STRING*)inst->fbDatObjCreate.pDatObjMem;
				inst->pTextEnd = inst->pTextStart + inst->fbDatObjCreate.len;
				inst->pText = inst->pTextStart;
				inst->eStep = eSTEP_READ_FILE;
			}
			else if(inst->fbDatObjCreate.status != eBRB_ERR_BUSY)
			{
				// Fehler merken
				inst->nStatusIntern = inst->fbDatObjCreate.status;
				// Datei muß auf jeden Fall geschlossen werden
				inst->eStep = eSTEP_CLOSE_FILE;
			}
			break;

		case eSTEP_READ_FILE:
			// Datei in das Datenobjekt einlesen
			inst->nStatus = eBRB_ERR_BUSY;
			inst->fbFileRead.enable = 1;
			inst->fbFileRead.ident = inst->fbFileOpen.ident;
			inst->fbFileRead.offset = 0;
			inst->fbFileRead.pDest = inst->fbDatObjCreate.pDatObjMem;
			inst->fbFileRead.len = inst->fbFileOpen.filelen;
			FileRead(&inst->fbFileRead);
			if(inst->fbFileRead.status == 0)
			{
				inst->eStep = eSTEP_CLOSE_FILE;
			}
			else if(inst->fbFileRead.status != eBRB_ERR_BUSY)
			{
				// Fehler merken
				inst->nStatusIntern = inst->fbFileRead.status;
				// Datei muß auf jeden Fall geschlossen werden
				inst->eStep = eSTEP_CLOSE_FILE;
			}
			break;

		case eSTEP_CLOSE_FILE:
			// Datei schliessen
			inst->nStatus = eBRB_ERR_BUSY;
			inst->fbFileClose.enable = 1;
			inst->fbFileClose.ident = inst->fbFileOpen.ident;
			FileClose(&inst->fbFileClose);
			if(inst->fbFileClose.status == 0)
			{
				// Prüfen, ob vorher schon ein Fehler aufgetreten ist
				if(inst->nStatusIntern > 0)
				{
					// Datenobjekt muß auf jeden Fall gelöscht werden
					inst->eStep = eSTEP_DELETE_DATAOBJ_END;
				}
				else
				{
					inst->eStep = eSTEP_READ_LINES;
				}
			}
			else if(inst->fbFileClose.status != eBRB_ERR_BUSY)
			{
				// Prüfen, ob vorher schon ein Fehler aufgetreten ist
				if(inst->nStatusIntern > 0)
				{
					// Datenobjekt muß auf jeden Fall gelöscht werden
					inst->eStep = eSTEP_DELETE_DATAOBJ_END;
				}
				else
				{
					// Fehler merken
					inst->nStatusIntern = inst->fbFileClose.status;
					// Datenobjekt muß auf jeden Fall gelöscht werden
					inst->eStep = eSTEP_DELETE_DATAOBJ_END;
				}
			}
			break;

		case eSTEP_READ_LINES:
			inst->nStatus = eBRB_ERR_BUSY;
			inst->nLineCountRead = 0;
			do
			{
				if(BrbStringStartsWith(inst->pText, "//"))
				{
					// Kommentare werden überlesen
				}
				else
				{
					// Variable lesen
					BrbPvInfo_TYP PvInfo;
					memset(&PvInfo, 0, sizeof(PvInfo));
					STRING sPvValue[nBRB_PVNAME_CHAR_MAX];
					memset(&sPvValue, 0, sizeof(sPvValue));
					// Namen lesen
					inst->pText = ReadPvName(inst->pText, PvInfo.sName, inst->pTextEnd);
					if(inst->pText != 0)
					{
						// Wert lesen
						inst->pText = ReadPvValue(inst->pText, sPvValue, inst->pTextEnd);
						if(inst->pText != 0)
						{
							SetValue(&PvInfo, sPvValue);
						}
					}
				}
				// Auf den Anfang der nächsten Zeile springen
				inst->pText = SetToNextLine(inst->pText, inst->pTextEnd, (STRING*)&inst->sLineBreak);
				inst->nLineCountRead += 1;
				if((inst->pText >= inst->pTextEnd) || (inst->pText == 0))
				{
					// Ende der Datei erreicht -> Schleife verlassen
					inst->nLineCountRead = inst->nLinesToReadAtOneStep + 1;
					inst->eStep = eSTEP_DELETE_DATAOBJ_END;
					break;
				}
			}
			while(inst->nLineCountRead <= inst->nLinesToReadAtOneStep);
			break;

		case eSTEP_DELETE_DATAOBJ_END:
			// Datenobjekt löschen
			inst->nStatus = eBRB_ERR_BUSY;
			inst->fbDatObjDelete.enable = 1;
			inst->fbDatObjDelete.ident = inst->fbDatObjCreate.ident;
			DatObjDelete(&inst->fbDatObjDelete);
			if(inst->fbDatObjDelete.status != eBRB_ERR_BUSY)
			{
				if(inst->nStatusIntern > 0)
				{
					inst->nStatus = inst->nStatusIntern;
				}
				else
				{
					inst->nStatus = 0;
				}
				inst->eStep = eSTEP_INIT;
			}
			break;

	}
}

// Gibt die Adresse nach dem nächsten Zeilenumbruch zurück.
// 0, wenn es nicht gefunden wird.
STRING* SetToNextLine(STRING* pText, STRING* pTextEnd, STRING* pLineBreak)
{
	STRING* pResult = 0;
	if(pText != 0)
	{
		// Nach Zeilenumbruch suchen
		pResult = BrbStringGetAdrOf(pText, pLineBreak, (UDINT)(pTextEnd - pText));
		if(pResult >= pText)
		{
			// Gefunden -> CrLf überspringen
			pResult += 2;
		}
	}
	return pResult;
}

// Liest den Text bis zum nächsten = und gibt die Adresse danach zurück.
// 0, wenn es nicht gefunden wird.
STRING* ReadPvName(STRING* pText, STRING* pPvName, STRING* pTextEnd)
{
	STRING* pResult = 0;
	// Nach = suchen
	pResult = BrbStringGetAdrOf(pText, "=", (UDINT)(pTextEnd - pText));
	if(pResult >= pText)
	{
		// Gefunden -> Überspringen
		memcpy(pPvName, pText, (UDINT)(pResult - pText));
		pResult += 1;
	}
	return pResult;
}

// Liest den Text bis zum nächsten CrLf und gibt die Adresse zurück.
// 0, wenn es nicht gefunden wird.
STRING* ReadPvValue(STRING* pText, STRING* pPvValue, STRING* pTextEnd)
{
	STRING* pResult = 0;
	// Nach CrLf suchen
	pResult = BrbStringGetAdrOf(pText, "\r\n", (UDINT)(pTextEnd - pText));
	if(pResult >= pText)
	{

		// Gefunden -> Länge des Werts prüfen
		UDINT nLenValue = (UDINT)(pResult - pText);
		if(nLenValue >= nBRB_PVNAME_CHAR_MAX)
		{
			// Länge begrenzen
			nLenValue = nBRB_PVNAME_CHAR_MAX - 1;
		}
		// Wert kopieren
		memcpy(pPvValue, pText, nLenValue);
		// CrLf nicht überspringen (wird zum Erkennen der nächsten Zeile gebraucht)
	}
	return pResult;
}

// Setzt den Wert einer Pv als String.
void SetValue(BrbPvInfo_TYP* pPvInfo, STRING* pValue)
{
	UINT	nFuncStatus = 0;
	UDINT nLen = 0;
	STRING sItoA[20];
	memset(sItoA, 0, sizeof(sItoA));
	// Adresse der Variablen holen
	nFuncStatus = PV_xgetadr(pPvInfo->sName, &pPvInfo->nAdr, &nLen);
	if(nFuncStatus == 0)
	{
		// Datentyp der Variable holen
		nFuncStatus = PV_ninfo(pPvInfo->sName, &pPvInfo->nDataType, &pPvInfo->nLen, &pPvInfo->nDimension);
		if(nFuncStatus == 0)
		{
			// Wert in Datentyp wandeln und an der Adresse setzen
			switch(pPvInfo->nDataType)
			{
				case eDATATYPE_BOOL:
					{
						DINT nValue = brsatoi((UDINT)pValue);
						*(BOOL*)pPvInfo->nAdr = (BOOL)nValue;
					}
					break;

				case eDATATYPE_SINT:
					{
						DINT nValue = brsatoi((UDINT)pValue);
						*(SINT*)pPvInfo->nAdr = (SINT)nValue;
					}
					break;

				case eDATATYPE_INT:
					{
						DINT nValue = brsatoi((UDINT)pValue);
						*(INT*)pPvInfo->nAdr = (INT)nValue;
					}
					break;

				case eDATATYPE_DINT:
					{
						DINT nValue = brsatoi((UDINT)pValue);
						*(DINT*)pPvInfo->nAdr = (DINT)nValue;
					}
					break;

				case eDATATYPE_USINT:
					{
						DINT nValue = brsatoi((UDINT)pValue);
						*(USINT*)pPvInfo->nAdr = (USINT)nValue;
					}
					break;

				case eDATATYPE_UINT:
					{
						DINT nValue = brsatoi((UDINT)pValue);
						*(UINT*)pPvInfo->nAdr = (UINT)nValue;
					}
					break;

				case eDATATYPE_UDINT:
					{
						UDINT nValue = BrbAsciiToUdint(pValue);
						*(UDINT*)pPvInfo->nAdr = (UDINT)nValue;
					}
					break;

				case eDATATYPE_REAL:
					{
						REAL rValue = brsatof((UDINT)pValue);
						*(REAL*)pPvInfo->nAdr = (REAL)rValue;
					}
					break;

				case eDATATYPE_STRING:
					{
						strcpy((STRING*)pPvInfo->nAdr, pValue); // NOLINT(clang-analyzer-security.insecureAPI.strcpy)
					}
					break;

				case eDATATYPE_DATE_AND_TIME:
					{
						UDINT nValue = BrbAsciiToUdint(pValue);
						*(UDINT*)pPvInfo->nAdr = (UDINT)nValue;
					}
					break;

				case eDATATYPE_TIME:
					{
						DINT nValue = brsatoi((UDINT)pValue);
						*(DINT*)pPvInfo->nAdr = (DINT)nValue;
					}
					break;

			}
		}
	}
}

// NOLINTEND(readability-*, bugprone-easily-swappable-parameters, clang-diagnostic-invalid-utf8, clang-diagnostic-invalid-source-encoding, clang-diagnostic-pointer-arith, clang-diagnostic-strict-prototypes, hicpp-uppercase-literal-suffix, cppcoreguidelines-*, performance-*)
```

#### BrbLoadVarBin.c
```c
/********************************************************************
 * COPYRIGHT -- Bernecker + Rainer
 ********************************************************************
 * Library: BrbLib
 * File: BrbLoadVarBin.c
 * Author: niedermeierr
 * Created: June 11, 2013
 ********************************************************************
 * Implementation of library BrbLib
 ********************************************************************/

#include <bur/plctypes.h>
#ifdef __cplusplus
	extern "C"
	{
#endif

#include "BrbLib.h"
#include <string.h>

#ifdef __cplusplus
	};
#endif

// NOLINTBEGIN(readability-*, bugprone-easily-swappable-parameters, clang-diagnostic-invalid-utf8, clang-diagnostic-invalid-source-encoding, clang-diagnostic-pointer-arith, clang-diagnostic-strict-prototypes, hicpp-uppercase-literal-suffix, cppcoreguidelines-*, performance-*)

// Eigene Enums und Typen
enum Steps_ENUM
{
	eSTEP_INIT,
	eSTEP_OPEN_FILE,
	eSTEP_TEST_SIZE,
	eSTEP_READ_FILE,
	eSTEP_CLOSE_FILE,
};

/* Lädt eine Binär-Datei mit Variablen-Werten */
void BrbLoadVarBin(struct BrbLoadVarBin* inst) // NOLINT(readability-function-cognitive-complexity)
{
	// Prüfung der Parameter
	if(inst->pDevice == 0)
	{
		inst->nStatus = eBRB_ERR_NULL_POINTER;
		return;
	}
	if(inst->pFile == 0)
	{
		inst->nStatus = eBRB_ERR_NULL_POINTER;
		return;
	}

	UINT	nFuncStatus = 0;
	switch(inst->eStep)
	{
		case eSTEP_INIT:
			// Fub initialisieren
			inst->nStatus = eBRB_ERR_BUSY;
			inst->nStatusIntern = 0;
			memset(&inst->fbFileOpen, 0, sizeof(inst->fbFileOpen));
			memset(&inst->PvInfo, 0, sizeof(inst->PvInfo));
			memset(&inst->fbFileRead, 0, sizeof(inst->fbFileRead));
			memset(&inst->fbFileClose, 0, sizeof(inst->fbFileClose));
			inst->eStep = eSTEP_OPEN_FILE;
			break;

		case eSTEP_OPEN_FILE:
			// Datei öffnen
			inst->nStatus = eBRB_ERR_BUSY;
			inst->fbFileOpen.enable = 1;
			inst->fbFileOpen.pDevice = (UDINT)inst->pDevice;
			inst->fbFileOpen.pFile = (UDINT)inst->pFile;
			FileOpen(&inst->fbFileOpen);
			if(inst->fbFileOpen.status == 0)
			{
				inst->eStep = eSTEP_TEST_SIZE;
			}
			else if(inst->fbFileOpen.status != eBRB_ERR_BUSY)
			{
				inst->nStatus = inst->fbFileOpen.status;
				inst->eStep = eSTEP_INIT;
			}
			break;

		case eSTEP_TEST_SIZE:
			// Prüfen, ob die Dateigröße zur Größe der Variable passt
			inst->nStatus = eBRB_ERR_BUSY;
			// Adresse der Variable holen
			nFuncStatus = PV_xgetadr((STRING*)inst->pVarName, &inst->PvInfo.nAdr, &inst->PvInfo.nLen);
			if(nFuncStatus == 0)
			{
				// Größe der Variable holen
				nFuncStatus = PV_ninfo((STRING*)inst->pVarName, &inst->PvInfo.nDataType, &inst->PvInfo.nLen, &inst->PvInfo.nDimension);
				if(nFuncStatus == 0)
				{
					if(inst->bAllowBiggerVar == 1)
					{
						if(inst->PvInfo.nLen >= inst->fbFileOpen.filelen)
						{
							inst->eStep = eSTEP_READ_FILE;
						}
						else
						{
							// Fehler merken
							inst->nStatusIntern = ERR_BUR_ILLLEN; // = Ungültige Längenangabe
							// Datei muß auf jeden Fall geschlossen werden
							inst->eStep = eSTEP_CLOSE_FILE;
						}
					}
					else
					{
						if(inst->PvInfo.nLen == inst->fbFileOpen.filelen)
						{
							inst->eStep = eSTEP_READ_FILE;
						}
						else
						{
							// Fehler merken
							inst->nStatusIntern = ERR_BUR_ILLLEN; // = Ungültige Längenangabe
							// Datei muß auf jeden Fall geschlossen werden
							inst->eStep = eSTEP_CLOSE_FILE;
						}
					}
				}
				else
				{
					// Fehler merken
					inst->nStatusIntern = nFuncStatus;
					// Datei muß auf jeden Fall geschlossen werden
					inst->eStep = eSTEP_CLOSE_FILE;
				}
			}
			else
			{
				// Fehler merken
				inst->nStatusIntern = nFuncStatus;
				// Datei muß auf jeden Fall geschlossen werden
				inst->eStep = eSTEP_CLOSE_FILE;
			}
			break;

		case eSTEP_READ_FILE:
			// Einlesen der Datei auf die Variablen-Adresse
			inst->nStatus = eBRB_ERR_BUSY;
			inst->fbFileRead.enable = 1;
			inst->fbFileRead.ident = inst->fbFileOpen.ident;
			inst->fbFileRead.offset = 0;
			inst->fbFileRead.pDest = inst->PvInfo.nAdr;
			inst->fbFileRead.len = inst->PvInfo.nLen;
			FileRead(&inst->fbFileRead);
			if(inst->fbFileRead.status == 0)
			{
				inst->eStep = eSTEP_CLOSE_FILE;
			}
			else if(inst->fbFileRead.status != eBRB_ERR_BUSY)
			{
				// Fehler merken
				inst->nStatusIntern = inst->fbFileRead.status;
				// Datei muß auf jeden Fall geschlossen werden
				inst->eStep = eSTEP_CLOSE_FILE;
			}
			break;

		case eSTEP_CLOSE_FILE:
			// Datei schliessen
			inst->nStatus = eBRB_ERR_BUSY;
			inst->fbFileClose.enable = 1;
			inst->fbFileClose.ident = inst->fbFileOpen.ident;
			FileClose(&inst->fbFileClose);
			if(inst->fbFileClose.status == 0)
			{
				// Prüfen, ob vorher schon ein Fehler aufgetreten ist
				if(inst->nStatusIntern > 0)
				{
					inst->nStatus = inst->nStatusIntern;
					inst->eStep = eSTEP_INIT;
				}
				else
				{
					inst->nStatus = 0;
					inst->eStep = eSTEP_INIT;
				}
			}
			else if(inst->fbFileClose.status != eBRB_ERR_BUSY)
			{
				// Prüfen, ob vorher schon ein Fehler aufgetreten ist
				if(inst->nStatusIntern > 0)
				{
					inst->nStatus = inst->nStatusIntern;
					inst->eStep = eSTEP_INIT;
				}
				else
				{
					inst->nStatus = inst->fbFileClose.status;
					inst->eStep = eSTEP_INIT;
				}
			}
			break;

	}
}

// NOLINTEND(readability-*, bugprone-easily-swappable-parameters, clang-diagnostic-invalid-utf8, clang-diagnostic-invalid-source-encoding, clang-diagnostic-pointer-arith, clang-diagnostic-strict-prototypes, hicpp-uppercase-literal-suffix, cppcoreguidelines-*, performance-*)
```

#### BrbSaveVarAscii.c
```c
/********************************************************************
 * COPYRIGHT -- Bernecker + Rainer
 ********************************************************************
 * Library: BrbLib
 * File: BrbSaveVarAscii.c
 * Author: niedermeierr
 * Created: June 11, 2013
 ********************************************************************
 * Implementation of library BrbLib
 ********************************************************************/

#include <bur/plctypes.h>
#ifdef __cplusplus
	extern "C"
	{
#endif

#include "BrbLib.h"
#include <string.h>
#include <AnsiCFunc.h>

#ifdef __cplusplus
	};
#endif

// NOLINTBEGIN(readability-*, bugprone-easily-swappable-parameters, clang-diagnostic-invalid-utf8, clang-diagnostic-invalid-source-encoding, clang-diagnostic-pointer-arith, clang-diagnostic-strict-prototypes, hicpp-uppercase-literal-suffix, cppcoreguidelines-*, performance-*, clang-analyzer-security.insecureAPI.strcpy)

// Eigene Enums und Typen
enum Steps_ENUM
{
	eSTEP_INIT,
	eSTEP_DELETE_FILE,
	eSTEP_CREATE_FILE,
	eSTEP_GET_HEADER,
	eSTEP_SET_ROOT_PV,
	eSTEP_GET_LINES,
	eSTEP_WRITE_LINES,
	eSTEP_CLOSE_FILE
};

enum Datatypes_ENUM
{
	eDATATYPE_STRUCT,
	eDATATYPE_BOOL,
	eDATATYPE_SINT,
	eDATATYPE_INT,
	eDATATYPE_DINT,
	eDATATYPE_USINT,
	eDATATYPE_UINT,
	eDATATYPE_UDINT,
	eDATATYPE_REAL,
	eDATATYPE_STRING,
	eDATATYPE_DATE_AND_TIME = 11,
	eDATATYPE_TIME,
	eDATATYPE_STRUCT_ARRAY = 15
};

// Prototypen
void GetValue(BrbPvInfo_TYP* pPvInfo, STRING* pValue);

/* Speichert eine Variable mit allen Elementen in einer Ascii-Datei */
void BrbSaveVarAscii(struct BrbSaveVarAscii* inst) // NOLINT(readability-function-cognitive-complexity)
{
	// Prüfung der Parameter
	if(inst->pDevice == 0)
	{
		inst->nStatus = eBRB_ERR_NULL_POINTER;
		return;
	}
	if(inst->pFile == 0)
	{
		inst->nStatus = eBRB_ERR_NULL_POINTER;
		return;
	}
	if(inst->pVarName == 0)
	{
		inst->nStatus = eBRB_ERR_NULL_POINTER;
		return;
	}

	UINT	nFuncStatus = 0;
	STRING sValue[1000];
	STRING sName[40];
	STRING sIndex[20];

	switch(inst->eStep)
	{
		case eSTEP_INIT:
			// Fub initialisieren
			inst->nStatus = eBRB_ERR_BUSY;
			inst->nStatusIntern = 0;
			memset(&inst->fbFileDelete, 0, sizeof(inst->fbFileDelete));
			memset(&inst->fbFileCreate, 0, sizeof(inst->fbFileCreate));
			inst->nOffset = 0;
			inst->nLineCountWrite = 0;
			inst->nCharCountMaxPerWrite = 0;
			memset(&inst->fbFileWrite, 0, sizeof(inst->fbFileWrite));
			memset(&inst->fbFileClose, 0, sizeof(inst->fbFileClose));
			if(inst->nLinesToWriteAtOneStep == 0)
			{
				// Wenn keine Anzahl angegeben ist, einen Defaultwert verwenden
				inst->nLinesToWriteAtOneStep = 10;
			}
			inst->bVarFinished = 0;
			inst->eStep = eSTEP_DELETE_FILE;
			break;

		case eSTEP_DELETE_FILE:
			// Evtl. vorhandene Datei löschen
			inst->nStatus = eBRB_ERR_BUSY;
			inst->fbFileDelete.enable = 1;
			inst->fbFileDelete.pDevice = (UDINT)inst->pDevice;
			inst->fbFileDelete.pName = (UDINT)inst->pFile;
			FileDelete(&inst->fbFileDelete);
			if(inst->fbFileDelete.status != eBRB_ERR_BUSY)
			{
				inst->eStep = eSTEP_CREATE_FILE;
			}
			break;

		case eSTEP_CREATE_FILE:
			// Datei neu erzeugen
			inst->nStatus = eBRB_ERR_BUSY;
			inst->fbFileCreate.enable = 1;
			inst->fbFileCreate.pDevice = (UDINT)inst->pDevice;
			inst->fbFileCreate.pFile = (UDINT)inst->pFile;
			FileCreate(&inst->fbFileCreate);
			if(inst->fbFileCreate.status == 0)
			{
				inst->eStep = eSTEP_GET_HEADER;
			}
			else if(inst->fbFileCreate.status != eBRB_ERR_BUSY)
			{
				inst->nStatus = inst->fbFileCreate.status;
				inst->eStep = eSTEP_INIT;
			}
			break;

		case eSTEP_GET_HEADER:
			// Header erzeugen
			inst->nStatus = eBRB_ERR_BUSY;
			memset(&inst->sLines, 0, sizeof(inst->sLines));
			strcpy(inst->sLines, "// Parameterfile '");
			strcat(inst->sLines, (STRING*)inst->pFile);
			strcat(inst->sLines, "'\r\n");
			inst->nLineCountWrite += 1;
			strcat(inst->sLines, "// Variable: '");
			strcat(inst->sLines, (STRING*)inst->pVarName);
			strcat(inst->sLines, "'\r\n");
			inst->nLineCountWrite += 1;
			BrbGetCurrentTimeText(inst->sHelp, sizeof(inst->sHelp), "yyyy.mm.dd hh:MM:ss");
			strcat(inst->sLines, "// Date: ");
			strcat(inst->sLines, (STRING*)inst->sHelp);
			strcat(inst->sLines, "\r\n");
			inst->nLineCountWrite += 1;
			inst->eStep = eSTEP_SET_ROOT_PV;
			break;

		case eSTEP_SET_ROOT_PV:
			// Informationen der Basis-Pv holen
			inst->nStatus = eBRB_ERR_BUSY;
			memset(&inst->PvInfo, 0, sizeof(inst->PvInfo));
			inst->nPvLevel = 0;
			BrbStringCopy(inst->PvInfo[inst->nPvLevel].sName, (STRING*)inst->pVarName, sizeof(inst->PvInfo[inst->nPvLevel].sName));
			inst->eStep = eSTEP_GET_LINES;
			break;

		case eSTEP_GET_LINES:
			// Die Zeilen der Elemente erzeugen
			inst->nStatus = eBRB_ERR_BUSY;
			do
			{
				// Prüfen, ob die Information des aktuellen Elements schon geholt wurden
				nFuncStatus = 0;
				if(inst->PvInfo[inst->nPvLevel].nLen == 0)
				{
					// Information des aktuellen Elements holen
					nFuncStatus = PV_ninfo((STRING*)&inst->PvInfo[inst->nPvLevel].sName, &inst->PvInfo[inst->nPvLevel].nDataType, &inst->PvInfo[inst->nPvLevel].nLen, &inst->PvInfo[inst->nPvLevel].nDimension);
				}
				if(nFuncStatus != 0)
				{
					inst->nStatusIntern = nFuncStatus;
					inst->bVarFinished = 1;
				}
				else
				{
					// Datentyp und Feldgröße prüfen
					if(inst->PvInfo[inst->nPvLevel].nDataType == eDATATYPE_STRUCT_ARRAY)
					{
						// Struktur-Array
						if(inst->PvInfo[inst->nPvLevel].nItemIndex < inst->PvInfo[inst->nPvLevel].nDimension)
						{
							// Nächstes Level
							inst->nPvLevel += 1;
							memset(&inst->PvInfo[inst->nPvLevel], 0, sizeof(inst->PvInfo[inst->nPvLevel]));
							// Namen zusammensetzen
							// "Root.StructArray.StructArray[x]"
							BrbStringCat(inst->PvInfo[inst->nPvLevel].sName, inst->PvInfo[inst->nPvLevel-1].sName, sizeof(inst->PvInfo[inst->nPvLevel].sName));
							BrbStringCat(inst->PvInfo[inst->nPvLevel].sName, "[", sizeof(inst->PvInfo[inst->nPvLevel].sName));
							brsitoa((DINT)inst->PvInfo[inst->nPvLevel-1].nItemIndex, (UDINT)&sIndex);
							BrbStringCat(inst->PvInfo[inst->nPvLevel].sName, sIndex, sizeof(inst->PvInfo[inst->nPvLevel].sName));
							BrbStringCat(inst->PvInfo[inst->nPvLevel].sName, "]", sizeof(inst->PvInfo[inst->nPvLevel].sName));
						}
						else
						{
							// Array-Dimension erreicht
							if(inst->nPvLevel > 0)
							{
								// Vorheriges Level und nächstes Element
								inst->nPvLevel -= 1;
								inst->PvInfo[inst->nPvLevel].nItemIndex += 1;
							}
							else
							{
								// Alle Elemente der Basis-Pv durchlaufen
								inst->bVarFinished = 1;
							}
						}
					}
					else if(inst->PvInfo[inst->nPvLevel].nDataType == eDATATYPE_STRUCT)
					{
						// Einfache Struktur -> Element-Informationen holen
						nFuncStatus = PV_item(inst->PvInfo[inst->nPvLevel].sName, inst->PvInfo[inst->nPvLevel].nItemIndex, sName);
						if(nFuncStatus == 0)
						{
							// Element gültig -> Nächstes Level
							inst->nPvLevel += 1;
							memset(&inst->PvInfo[inst->nPvLevel], 0, sizeof(inst->PvInfo[inst->nPvLevel]));
							// Namen zusammensetzen
							// "Root.Element"
							BrbStringCat(inst->PvInfo[inst->nPvLevel].sName, inst->PvInfo[inst->nPvLevel-1].sName, sizeof(inst->PvInfo[inst->nPvLevel].sName));
							BrbStringCat(inst->PvInfo[inst->nPvLevel].sName, ".", sizeof(inst->PvInfo[inst->nPvLevel].sName));
							BrbStringCat(inst->PvInfo[inst->nPvLevel].sName, sName, sizeof(inst->PvInfo[inst->nPvLevel].sName));
						}
						else
						{
							// Keine weiteren Elemente
							if(inst->nPvLevel > 0)
							{
								// Vorheriges Level und nächstes Element
								memset(&inst->PvInfo[inst->nPvLevel], 0, sizeof(inst->PvInfo[inst->nPvLevel]));
								inst->nPvLevel -= 1;
								inst->PvInfo[inst->nPvLevel].nItemIndex += 1;
							}
							else
							{
								// Alle Elemente der Basis-Pv durchlaufen
								inst->bVarFinished = 1;
							}
						}
					}
					else
					{
						// Einfacher Datentyp
						if(inst->PvInfo[inst->nPvLevel].nDimension > 1)
						{
							// Einfaches Array
							// Prüfen, ob schon alle Felder durchlaufen sind
							if(inst->PvInfo[inst->nPvLevel].nItemIndex < inst->PvInfo[inst->nPvLevel].nDimension)
							{
								// Noch Felder übrig -> Nächstes Level
								inst->nPvLevel += 1;
								memset(&inst->PvInfo[inst->nPvLevel], 0, sizeof(inst->PvInfo[inst->nPvLevel]));
								// Namen zusammensetzen
								// "Root.Array.Array[x]"
								BrbStringCat(inst->PvInfo[inst->nPvLevel].sName, inst->PvInfo[inst->nPvLevel-1].sName, sizeof(inst->PvInfo[inst->nPvLevel].sName));
								BrbStringCat(inst->PvInfo[inst->nPvLevel].sName, "[", sizeof(inst->PvInfo[inst->nPvLevel].sName));
								brsitoa((DINT)inst->PvInfo[inst->nPvLevel-1].nItemIndex, (UDINT)&sIndex);
								BrbStringCat(inst->PvInfo[inst->nPvLevel].sName, sIndex, sizeof(inst->PvInfo[inst->nPvLevel].sName));
								BrbStringCat(inst->PvInfo[inst->nPvLevel].sName, "]", sizeof(inst->PvInfo[inst->nPvLevel].sName));
							}
							else
							{
								// Kein Feld übrig
								if(inst->nPvLevel > 0)
								{
									// Vorheriges Level und nächstes Element
									memset(&inst->PvInfo[inst->nPvLevel], 0, sizeof(inst->PvInfo[inst->nPvLevel]));
									inst->nPvLevel -= 1;
									inst->PvInfo[inst->nPvLevel].nItemIndex += 1;
								}
								else
								{
									// Alle Elemente der Basis-Pv durchlaufen
									inst->bVarFinished = 1;
								}
							}
						}
						else
						{
							// Einfacher Datentyp -> Zeile erzeugen
							// "PvName=Wert"
							strcat(inst->sLines, inst->PvInfo[inst->nPvLevel].sName);
							strcat(inst->sLines, "=");
							memset(&sValue, 0, sizeof(sValue));
							GetValue(&inst->PvInfo[inst->nPvLevel], sValue);
							strcat(inst->sLines, sValue);
							strcat(inst->sLines, "\r\n");
							inst->nLineCountWrite += 1;
							if(inst->nPvLevel > 0)
							{
								// Vorheriges Level und nächstes Element
								memset(&inst->PvInfo[inst->nPvLevel], 0, sizeof(inst->PvInfo[inst->nPvLevel]));
								inst->nPvLevel -= 1;
								inst->PvInfo[inst->nPvLevel].nItemIndex += 1;
							}
							else
							{
								// Nächstes Element
								inst->PvInfo[inst->nPvLevel].nItemIndex += 1;
							}
						}
					}
				}
			} while((inst->bVarFinished == 0) && (inst->nLineCountWrite < inst->nLinesToWriteAtOneStep));
			inst->eStep = eSTEP_WRITE_LINES;
			break;

		case eSTEP_WRITE_LINES:
			// Bisher erzeugte Zeilen schreiben
			inst->nStatus = eBRB_ERR_BUSY;
			inst->fbFileWrite.enable = 1;
			inst->fbFileWrite.ident = inst->fbFileCreate.ident;
			inst->fbFileWrite.offset = inst->nOffset;
			inst->fbFileWrite.pSrc = (UDINT)&inst->sLines;
			inst->fbFileWrite.len = strlen((STRING*)&inst->sLines);
			FileWrite(&inst->fbFileWrite);
			if(inst->fbFileWrite.status == 0)
			{
				inst->nOffset += inst->fbFileWrite.len;
				memset(&inst->sLines, 0, sizeof(inst->sLines));
				inst->nLineCountWrite = 0;
				// Prüfen, ob noch Zeilen zu erzeugen sind
				if(inst->bVarFinished == 0)
				{
					inst->eStep = eSTEP_GET_LINES;
				}
				else
				{
					inst->eStep = eSTEP_CLOSE_FILE;
				}
			}
			else if(inst->fbFileWrite.status != eBRB_ERR_BUSY)
			{
				// Fehler merken
				if(inst->nStatusIntern == 0)
				{
					inst->nStatusIntern = inst->fbFileWrite.status;
				}
				// Datei muß auf jeden Fall geschlossen werden
				inst->eStep = eSTEP_CLOSE_FILE;
			}
			// Den größten Wert für die Zeichen pro Zeile ermitteln
			if(inst->nCharCountMaxPerWrite < inst->fbFileWrite.len)
			{
				inst->nCharCountMaxPerWrite = inst->fbFileWrite.len;
			}
			break;

		case eSTEP_CLOSE_FILE:
			// Datei schliessen
			inst->nStatus = eBRB_ERR_BUSY;
			inst->fbFileClose.enable = 1;
			inst->fbFileClose.ident = inst->fbFileCreate.ident;
			FileClose(&inst->fbFileClose);
			if(inst->fbFileClose.status == 0)
			{
				// Prüfen, ob vorher schon ein Fehler aufgetreten ist
				if(inst->nStatusIntern > 0)
				{
					inst->nStatus = inst->nStatusIntern;
					inst->eStep = eSTEP_INIT;
				}
				else
				{
					inst->nStatus = 0;
					inst->eStep = eSTEP_INIT;
				}
			}
			else if(inst->fbFileClose.status != eBRB_ERR_BUSY)
			{
				// Prüfen, ob vorher schon ein Fehler aufgetreten ist
				if(inst->nStatusIntern > 0)
				{
					inst->nStatus = inst->nStatusIntern;
					inst->eStep = eSTEP_INIT;
				}
				else
				{
					inst->nStatus = inst->fbFileClose.status;
					inst->eStep = eSTEP_INIT;
				}
			}
			break;

	}
}

// Gibt den Wert einer Pv als String zurück.
void GetValue(BrbPvInfo_TYP* pPvInfo, STRING* pValue)
{
	// NOLINTBEGIN(clang-analyzer-security.insecureAPI.strcpy)
	UINT	nFuncStatus = 0;
	STRING sItoA[20];
	memset(sItoA, 0, sizeof(sItoA));
	// Adresse der Variable holen
	nFuncStatus = PV_xgetadr(pPvInfo->sName, &pPvInfo->nAdr, &pPvInfo->nLen);
	if(nFuncStatus == 0)
	{
		// Wert aufgrund des Datentyps an der Adresse holen und in String wandeln
		switch(pPvInfo->nDataType)
		{
			case eDATATYPE_BOOL:
				{
					BOOL bValue = *(BOOL*)pPvInfo->nAdr;
					brsitoa((DINT)bValue, (UDINT)&sItoA);
					strcpy(pValue, sItoA);
				}
				break;

			case eDATATYPE_SINT:
				{
					SINT nValue = *(SINT*)pPvInfo->nAdr;
					brsitoa((DINT)nValue, (UDINT)&sItoA);
					strcpy(pValue, sItoA);
				}
				break;

			case eDATATYPE_INT:
				{
					INT nValue = *(INT*)pPvInfo->nAdr;
					brsitoa((DINT)nValue, (UDINT)&sItoA);
					strcpy(pValue, sItoA);
				}
				break;

			case eDATATYPE_DINT:
				{
					DINT nValue = *(DINT*)pPvInfo->nAdr;
					brsitoa((DINT)nValue, (UDINT)&sItoA);
					strcpy(pValue, sItoA);
				}
				break;

			case eDATATYPE_USINT:
				{
					USINT nValue = *(USINT*)pPvInfo->nAdr;
					brsitoa((DINT)nValue, (UDINT)&sItoA);
					strcpy(pValue, sItoA);
				}
				break;

			case eDATATYPE_UINT:
				{
					UINT nValue = *(UINT*)pPvInfo->nAdr;
					brsitoa((DINT)nValue, (UDINT)&sItoA);
					strcpy(pValue, sItoA);
				}
				break;

			case eDATATYPE_UDINT:
				{
					UDINT nValue = *(UDINT*)pPvInfo->nAdr;
					BrbUdintToAscii(nValue, sItoA);
					strcpy(pValue, sItoA);
				}
				break;

			case eDATATYPE_REAL:
				{
					REAL rValue = *(REAL*)pPvInfo->nAdr;
					brsftoa(rValue, (UDINT)&sItoA);
					strcpy(pValue, sItoA);
				}
				break;

			case eDATATYPE_STRING:
				{
					strcpy(pValue, (STRING*)pPvInfo->nAdr);
				}
				break;

			case eDATATYPE_DATE_AND_TIME:
				{
					UDINT nValue = *(UDINT*)pPvInfo->nAdr;
					BrbUdintToAscii(nValue, sItoA);
					strcpy(pValue, sItoA);
				}
				break;

			case eDATATYPE_TIME:
				{
					DINT nValue = *(DINT*)pPvInfo->nAdr;
					brsitoa((DINT)nValue, (UDINT)&sItoA);
					strcpy(pValue, sItoA);
				}
				break;

		}
	}
	// NOLINTEND(clang-analyzer-security.insecureAPI.strcpy)
}

// NOLINTEND(readability-*, bugprone-easily-swappable-parameters, clang-diagnostic-invalid-utf8, clang-diagnostic-invalid-source-encoding, clang-diagnostic-pointer-arith, clang-diagnostic-strict-prototypes, hicpp-uppercase-literal-suffix, cppcoreguidelines-*, performance-*, clang-analyzer-security.insecureAPI.strcpy)
```

#### BrbSaveVarBin.c
```c
/********************************************************************
 * COPYRIGHT -- Bernecker + Rainer
 ********************************************************************
 * Library: BrbLib
 * File: BrbSaveVarBin.c
 * Author: niedermeierr
 * Created: June 11, 2013
 ********************************************************************
 * Implementation of library BrbLib
 ********************************************************************/

#include <bur/plctypes.h>
#ifdef __cplusplus
	extern "C"
	{
#endif

#include "BrbLib.h"
#include <string.h>

#ifdef __cplusplus
	};
#endif

// NOLINTBEGIN(readability-*, bugprone-easily-swappable-parameters, clang-diagnostic-invalid-utf8, clang-diagnostic-invalid-source-encoding, clang-diagnostic-pointer-arith, clang-diagnostic-strict-prototypes, hicpp-uppercase-literal-suffix, cppcoreguidelines-*, performance-*)

// Eigene Enums und Typen
enum Steps_ENUM
{
	eSTEP_INIT,
	eSTEP_GET_PV_INFO,
	eSTEP_DELETE_FILE,
	eSTEP_CREATE_FILE,
	eSTEP_WRITE_FILE,
	eSTEP_CLOSE_FILE,
};

/* Speichert eine Variable mit allen Elementen in einer Binär-Datei */
void BrbSaveVarBin(struct BrbSaveVarBin* inst) // NOLINT(readability-function-cognitive-complexity)
{
	// Prüfung der Parameter
	if(inst->pDevice == 0)
	{
		inst->nStatus = eBRB_ERR_NULL_POINTER;
		return;
	}
	if(inst->pFile == 0)
	{
		inst->nStatus = eBRB_ERR_NULL_POINTER;
		return;
	}
	if(inst->pVarName == 0)
	{
		inst->nStatus = eBRB_ERR_NULL_POINTER;
		return;
	}

	UINT	nFuncStatus = 0;
	switch(inst->eStep)
	{
		case eSTEP_INIT:
			// Fub initialisieren
			inst->nStatus = eBRB_ERR_BUSY;
			inst->nStatusIntern = 0;
			memset(&inst->PvInfo, 0, sizeof(inst->PvInfo));
			memset(&inst->fbFileDelete, 0, sizeof(inst->fbFileDelete));
			memset(&inst->fbFileCreate, 0, sizeof(inst->fbFileCreate));
			memset(&inst->fbFileWrite, 0, sizeof(inst->fbFileWrite));
			memset(&inst->fbFileClose, 0, sizeof(inst->fbFileClose));
			inst->eStep = eSTEP_GET_PV_INFO;
			break;

		case eSTEP_GET_PV_INFO:
			// Informationen der Variablen holen
			inst->nStatus = eBRB_ERR_BUSY;
			// Adresse der Variable holen
			nFuncStatus = PV_xgetadr((STRING*)inst->pVarName, &inst->PvInfo.nAdr, &inst->PvInfo.nLen);
			if(nFuncStatus == 0)
			{
				// Größe der Variable holen
				nFuncStatus = PV_ninfo((STRING*)inst->pVarName, &inst->PvInfo.nDataType, &inst->PvInfo.nLen, &inst->PvInfo.nDimension);
				if(nFuncStatus == 0)
				{
					inst->eStep = eSTEP_DELETE_FILE;
				}
				else
				{
					inst->nStatus = nFuncStatus;
					inst->eStep = eSTEP_INIT;
				}
			}
			else
			{
				inst->nStatus = nFuncStatus;
				inst->eStep = eSTEP_INIT;
			}
			break;

		case eSTEP_DELETE_FILE:
			// Evtl. vorhandene Datei löschen
			inst->nStatus = eBRB_ERR_BUSY;
			inst->fbFileDelete.enable = 1;
			inst->fbFileDelete.pDevice = (UDINT)inst->pDevice;
			inst->fbFileDelete.pName = (UDINT)inst->pFile;
			FileDelete(&inst->fbFileDelete);
			if(inst->fbFileDelete.status != eBRB_ERR_BUSY)
			{
				inst->eStep = eSTEP_CREATE_FILE;
			}
			break;

		case eSTEP_CREATE_FILE:
			// Datei neu erzeugen
			inst->nStatus = eBRB_ERR_BUSY;
			inst->fbFileCreate.enable = 1;
			inst->fbFileCreate.pDevice = (UDINT)inst->pDevice;
			inst->fbFileCreate.pFile = (UDINT)inst->pFile;
			FileCreate(&inst->fbFileCreate);
			if(inst->fbFileCreate.status == 0)
			{
				inst->eStep = eSTEP_WRITE_FILE;
			}
			else if(inst->fbFileCreate.status != eBRB_ERR_BUSY)
			{
				inst->nStatus = inst->fbFileCreate.status;
				inst->eStep = eSTEP_INIT;
			}
			break;

		case eSTEP_WRITE_FILE:
			// Speicher der Variable in die Datei schreiben
			inst->nStatus = eBRB_ERR_BUSY;
			inst->fbFileWrite.enable = 1;
			inst->fbFileWrite.ident = inst->fbFileCreate.ident;
			inst->fbFileWrite.offset = 0;
			inst->fbFileWrite.pSrc = (UDINT)inst->PvInfo.nAdr;
			inst->fbFileWrite.len = inst->PvInfo.nLen;
			FileWrite(&inst->fbFileWrite);
			if(inst->fbFileWrite.status == 0)
			{
				inst->eStep = eSTEP_CLOSE_FILE;
			}
			else if(inst->fbFileWrite.status != eBRB_ERR_BUSY)
			{
				// Fehler merken
				inst->nStatusIntern = inst->fbFileWrite.status;
				// Datei muß auf jeden Fall geschlossen werden
				inst->eStep = eSTEP_CLOSE_FILE;
			}
			break;

		case eSTEP_CLOSE_FILE:
			// Datei schliessen
			inst->nStatus = eBRB_ERR_BUSY;
			inst->fbFileClose.enable = 1;
			inst->fbFileClose.ident = inst->fbFileCreate.ident;
			FileClose(&inst->fbFileClose);
			if(inst->fbFileClose.status == 0)
			{
				// Prüfen, ob vorher schon ein Fehler aufgetreten ist
				if(inst->nStatusIntern > 0)
				{
					inst->nStatus = inst->nStatusIntern;
					inst->eStep = eSTEP_INIT;
				}
				else
				{
					inst->nStatus = 0;
					inst->eStep = eSTEP_INIT;
				}
			}
			else if(inst->fbFileClose.status != eBRB_ERR_BUSY)
			{
				// Prüfen, ob vorher schon ein Fehler aufgetreten ist
				if(inst->nStatusIntern > 0)
				{
					inst->nStatus = inst->nStatusIntern;
					inst->eStep = eSTEP_INIT;
				}
				else
				{
					inst->nStatus = inst->fbFileClose.status;
					inst->eStep = eSTEP_INIT;
				}
			}
			break;

	}
}

// NOLINTEND(readability-*, bugprone-easily-swappable-parameters, clang-diagnostic-invalid-utf8, clang-diagnostic-invalid-source-encoding, clang-diagnostic-pointer-arith, clang-diagnostic-strict-prototypes, hicpp-uppercase-literal-suffix, cppcoreguidelines-*, performance-*)
```

#### Package Logical/Libraries/BrbLib/FileHandling - Datei-Funktionen

#### BrbCheckUsbSticks.c - Prüft, ob ein Usb-Medium gesteckt wurde und linkt es
```c
/********************************************************************
 * COPYRIGHT -- Bernecker + Rainer
 ********************************************************************
 * Library: BrbLib
 * File: BrbCheckUsbSticks.c
 * Author: niedermeierr
 * Created: October 10, 2014
 ********************************************************************
 * Implementation of library BrbLib
 ********************************************************************/

#include <bur/plctypes.h>
#ifdef __cplusplus
	extern "C"
	{
#endif

#include "BrbLib.h"
#include <string.h>
#include <AnsiCFunc.h>

#ifdef __cplusplus
	};
#endif

// NOLINTBEGIN(readability-*, bugprone-easily-swappable-parameters, clang-diagnostic-invalid-utf8, clang-diagnostic-invalid-source-encoding, clang-diagnostic-pointer-arith, clang-diagnostic-strict-prototypes, hicpp-uppercase-literal-suffix, cppcoreguidelines-*, performance-*)

// Eigene Enums und Typen
enum Steps_ENUM
{
	eSTEP_INIT,
	eSTEP_CHECK_DEVICES,
	eSTEP_CHECK_UNLINK_DEVICES,
	eSTEP_REMOVE_DEVICE,
	eSTEP_UNLINK_DEVICE,
	eSTEP_CHECK_LINK_DEVICES,
	eSTEP_ADD_DEVICE,
	eSTEP_LINK_DEVICE,
};

/* Prüft, ob ein Usb-Medium gesteckt wurde und linkt es */
void BrbCheckUsbSticks(struct BrbCheckUsbSticks* inst) // NOLINT(readability-function-cognitive-complexity)
{
	switch(inst->eStep)
	{
		case eSTEP_INIT:
			// Fub initialisieren
			memset(&inst->fbUsbNodeGet, 0, sizeof(inst->fbUsbNodeGet));
			memset(&inst->UsbNodeInfo, 0, sizeof(inst->UsbNodeInfo));
			memset(&inst->DeviceListMan, 0, sizeof(inst->DeviceListMan));
			inst->DeviceListMan.pList = (UDINT)&inst->UsbDeviceList;
			inst->DeviceListMan.nEntryLength = sizeof(BrbUsbDeviceListEntry_TYP);
			inst->DeviceListMan.nIndexMax = nBRB_USB_DEVICE_LIST_INDEX_MAX;
			BrbMemListClear(&inst->DeviceListMan);
			inst->eStep = eSTEP_CHECK_DEVICES;
			break;

		case eSTEP_CHECK_DEVICES:
			inst->nStatus = 0;
			// Änderung prüfen
			inst->fbUsbNodeListGet.enable = 1;
			inst->fbUsbNodeListGet.pBuffer = (UDINT)&inst->UsbNodeList;
			inst->fbUsbNodeListGet.bufferSize = sizeof(inst->UsbNodeList);
			inst->fbUsbNodeListGet.filterInterfaceClass = asusb_CLASS_MASS_STORAGE;
			inst->fbUsbNodeListGet.filterInterfaceSubClass = asusb_SUBCLASS_SCSI_COMMAND_SET;
			UsbNodeListGet(&inst->fbUsbNodeListGet);
			if(inst->fbUsbNodeListGet.status == 0 || inst->fbUsbNodeListGet.status == asusbERR_USB_NOTFOUND)
			{
				if(inst->fbUsbNodeListGet.attachDetachCount != inst->nAttachDetachCountOld)
				{
					// Änderung erkannt
					inst->nStatus = eBRB_ERR_BUSY;
					inst->nUsbDeviceIndex = 0;
					inst->eStep = eSTEP_CHECK_UNLINK_DEVICES;
				}
				inst->nAttachDetachCountOld = inst->fbUsbNodeListGet.attachDetachCount;
			}
			else if(inst->fbUsbNodeListGet.status != eBRB_ERR_BUSY)
			{
				// Fehler
				inst->nStatus = inst->fbUsbNodeListGet.status;
			}
			inst->bUsbDeviceCountChanged = 0;
			break;

		case eSTEP_CHECK_UNLINK_DEVICES:
			// Prüfen, ob ein Device entfernt werden muss -> Liste der Devices durchtickern
			if(inst->nUsbDeviceIndex < inst->DeviceListMan.nEntryCount)
			{
				if(inst->UsbDeviceList[inst->nUsbDeviceIndex].nNode > 0)
				{
					// Prüfen, ob es den Node noch gibt
					BOOL bNodeFound = 0;
					for(inst->nUsbNodeIndex=0; inst->nUsbNodeIndex<=nBRB_USB_DEVICE_LIST_INDEX_MAX; inst->nUsbNodeIndex++)
					{
						if(inst->UsbDeviceList[inst->nUsbDeviceIndex].nNode == inst->UsbNodeList[inst->nUsbNodeIndex])
						{
							bNodeFound = 1;
							break;
						}
					}
					if(bNodeFound == 0)
					{
						// Node ist nicht mehr vorhanden -> Device löschen
						inst->eStep = eSTEP_REMOVE_DEVICE;
					}
					else
					{
						// Nächtes Device
						inst->nUsbDeviceIndex += 1;
					}
				}
			}
			else
			{
				// Device-Liste ist zu Ende
				inst->nUsbNodeIndex = 0;
				inst->eStep = eSTEP_CHECK_LINK_DEVICES;
			}
			break;

		case eSTEP_REMOVE_DEVICE:
			BrbMemListOut(&inst->DeviceListMan, inst->nUsbDeviceIndex, (UDINT)&inst->UsbDeviceListEntry);
			if(inst->UsbDeviceListEntry.nHandle > 0)
			{
				// Device muss ungelinkt werden
				inst->eStep = eSTEP_UNLINK_DEVICE;
			}
			else
			{
				// Nächtes Device
				inst->nUsbDeviceIndex += 1;
				inst->eStep = eSTEP_CHECK_UNLINK_DEVICES;
			}
			break;

		case eSTEP_UNLINK_DEVICE:
			inst->fbDevUnlink.enable = 1;
			inst->fbDevUnlink.handle = inst->UsbDeviceListEntry.nHandle;
			DevUnlink(&inst->fbDevUnlink);
			if(inst->fbDevUnlink.status != eBRB_ERR_BUSY)
			{
				// Nächtes Device
				inst->nUsbDeviceIndex += 1;
				inst->eStep = eSTEP_CHECK_UNLINK_DEVICES;
			}
			break;

		case eSTEP_CHECK_LINK_DEVICES:
			// Prüfen, ob ein Device hinzukommt -> Liste der Nodes durchtickern
			if(inst->nUsbNodeIndex <= nBRB_USB_DEVICE_LIST_INDEX_MAX)
			{
				if(inst->UsbNodeList[inst->nUsbNodeIndex] > 0)
				{
					// Prüfen, ob es das Device schon gibt
					BOOL bDeviceFound = 0;
					for(inst->nUsbDeviceIndex=0; inst->nUsbDeviceIndex<inst->DeviceListMan.nEntryCount; inst->nUsbDeviceIndex++)
					{
						if(inst->UsbDeviceList[inst->nUsbDeviceIndex].nNode == inst->UsbNodeList[inst->nUsbNodeIndex])
						{
							bDeviceFound = 1;
							break;
						}
					}
					if(bDeviceFound == 0)
					{
						// Device ist noch nicht vorhanden -> Device hinzufügen
						inst->eStep = eSTEP_ADD_DEVICE;
					}
					else
					{
						// Device ist schon vorhanden ->Nächster Node
						inst->nUsbNodeIndex += 1;
					}
				}
				else
				{
					// Nächster Node
					inst->nUsbNodeIndex += 1;
				}
			}
			else
			{
				// Liste ist zu Ende
				inst->nUsbDeviceCount = (UINT)inst->DeviceListMan.nEntryCount;
				inst->bUsbDeviceCountChanged = 1;
				inst->eStep = eSTEP_CHECK_DEVICES;
			}
			break;

		case eSTEP_ADD_DEVICE:
			// Informationen holen
			inst->fbUsbNodeGet.enable = 1;
			inst->fbUsbNodeGet.nodeId = inst->UsbNodeList[inst->nUsbNodeIndex];
			inst->fbUsbNodeGet.pBuffer = (UDINT)&inst->UsbNodeInfo;
			inst->fbUsbNodeGet.bufferSize = sizeof(inst->UsbNodeInfo);
			UsbNodeGet(&inst->fbUsbNodeGet);
			if(inst->fbUsbNodeGet.status == 0)
			{
				// Neues Device hinzufügen
				memset(&inst->UsbDeviceListEntry, 0, sizeof(inst->UsbDeviceListEntry));
				inst->UsbDeviceListEntry.nNode = inst->UsbNodeList[inst->nUsbNodeIndex];
				strncpy((STRING*)&inst->UsbDeviceListEntry.sInterfaceName, (STRING*)&inst->UsbNodeInfo.ifName, sizeof(inst->UsbDeviceListEntry.sInterfaceName));
				BrbStringCopy((STRING*)&inst->UsbDeviceListEntry.sDeviceName, "BrbUsb_", sizeof(inst->UsbDeviceListEntry.sDeviceName));
				BrbStringCat((STRING*)&inst->UsbDeviceListEntry.sDeviceName, (STRING*)&inst->UsbDeviceListEntry.sInterfaceName, sizeof(inst->UsbDeviceListEntry.sDeviceName));
				inst->nUsbDeviceIndex = (UINT)BrbMemListIn(&inst->DeviceListMan, inst->DeviceListMan.nEntryCount, (UDINT)&inst->UsbDeviceListEntry);
				if(inst->bAutoLink == 1)
				{
					// Device muss gelinkt werden
					memset(&inst->sLinkParameter, 0, sizeof(inst->sLinkParameter));
					BrbStringCopy((STRING*)&inst->sLinkParameter, "/DEVICE=", sizeof(inst->sLinkParameter));
					BrbStringCat((STRING*)&inst->sLinkParameter, (STRING*)&inst->UsbDeviceList[inst->nUsbNodeIndex].sInterfaceName, sizeof(inst->sLinkParameter));
					inst->eStep = eSTEP_LINK_DEVICE;
				}
				else
				{
					// Nächster Node
					inst->nUsbNodeIndex += 1;
					inst->eStep = eSTEP_CHECK_LINK_DEVICES;
				}
			}
			else if(inst->fbUsbNodeGet.status != eBRB_ERR_BUSY)
			{
				// Fehler (sollte nicht auftreten)
				// Nächster Node
				inst->nUsbNodeIndex += 1;
				inst->eStep = eSTEP_CHECK_LINK_DEVICES;
			}
			break;

		case eSTEP_LINK_DEVICE:
			inst->fbDevLink.enable = 1;
			inst->fbDevLink.pDevice = (UDINT)&inst->UsbDeviceListEntry.sDeviceName;
			inst->fbDevLink.pParam = (UDINT)&inst->sLinkParameter;
			DevLink(&inst->fbDevLink);
			if(inst->fbDevLink.status == 0)
			{
				inst->UsbDeviceList[inst->nUsbDeviceIndex].nHandle = inst->fbDevLink.handle;
				// Nächster Node
				inst->nUsbNodeIndex += 1;
				inst->eStep = eSTEP_CHECK_LINK_DEVICES;
			}
			else if(inst->fbDevLink.status == fiERR_DEVICE_ALREADY_EXIST)
			{
				inst->UsbDeviceList[inst->nUsbNodeIndex].nHandle = inst->fbDevLink.handle;
				// Nächster Node
				inst->nUsbNodeIndex += 1;
				inst->eStep = eSTEP_CHECK_LINK_DEVICES;
			}
			else if(inst->fbDevLink.status != eBRB_ERR_BUSY)
			{
				inst->UsbDeviceList[inst->nUsbNodeIndex].nHandle = 0;
				// Nächster Node
				inst->nUsbNodeIndex += 1;
				inst->eStep = eSTEP_CHECK_LINK_DEVICES;
			}
			break;

	}
}

// NOLINTEND(readability-*, bugprone-easily-swappable-parameters, clang-diagnostic-invalid-utf8, clang-diagnostic-invalid-source-encoding, clang-diagnostic-pointer-arith, clang-diagnostic-strict-prototypes, hicpp-uppercase-literal-suffix, cppcoreguidelines-*, performance-*)
```
